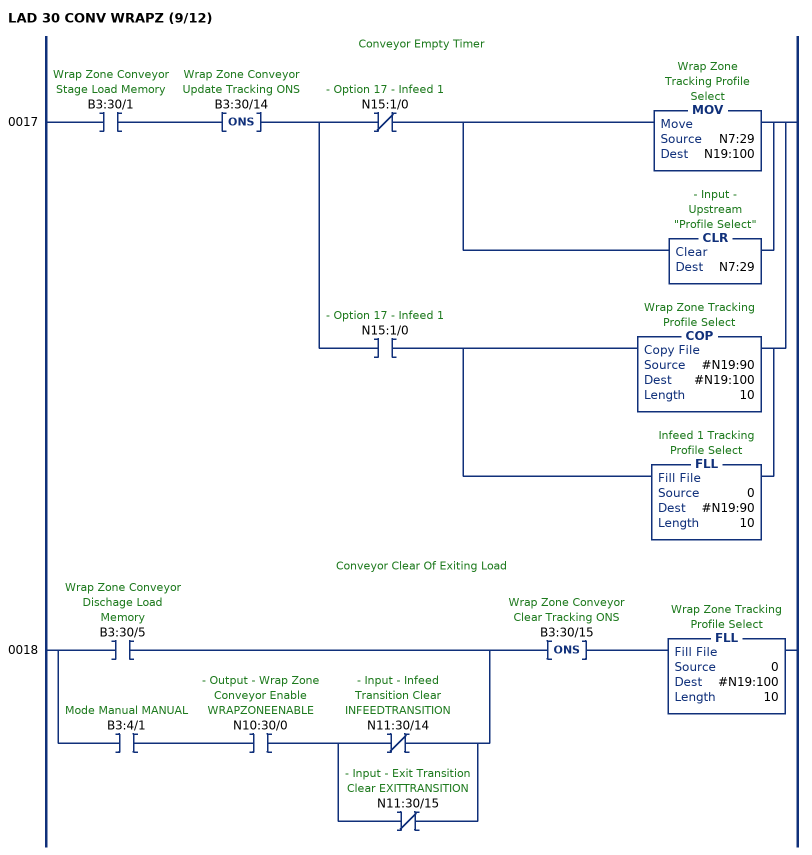
% Rung: 17 %
% Conveyor Empty Timer %
SOR XIC B3:30/1 ONS B3:30/14 BST XIO N15:1/0 BST MOV N7:29 N19:100 NXB CLR N7:29 BND NXB XIC N15:1/0 BST COP #N19:90 #N19:100 10 NXB FLL 0 #N19:90 10 BND BND EOR
%   B3:30/1  "Wrap Zone Conveyor Stage Load Memory" %
%   B3:30/14  "Wrap Zone Conveyor Update Tracking ONS" %
%   N15:1/0  "- Option 17 - Infeed 1" %
%   N7:29  "- Input - Upstream "Profile Select"" %
%   N19:100  "Wrap Zone Tracking Profile Select" %
%   N19:90  "Infeed 1 Tracking Profile Select" %
% Rung: 18 %
% Conveyor Clear Of Exiting Load %
SOR BST XIC B3:30/5 NXB XIC B3:4/1 XIC N10:30/0 BST XIO N11:30/14 NXB XIO N11:30/15 BND BND ONS B3:30/15 FLL 0 #N19:100 10 EOR
%   B3:30/5  "Wrap Zone Conveyor Dischage Load Memory" %
%   B3:4/1  MANUAL  "Mode Manual" %
%   N10:30/0  WRAPZONEENABLE  "- Output - Wrap Zone Conveyor Enable" %
%   N11:30/14  INFEEDTRANSITION  "- Input - Infeed Transition Clear" %
%   N11:30/15  EXITTRANSITION  "- Input - Exit Transition Clear" %
%   B3:30/15  "Wrap Zone Conveyor Clear Tracking ONS" %
%   N19:100  "Wrap Zone Tracking Profile Select" %

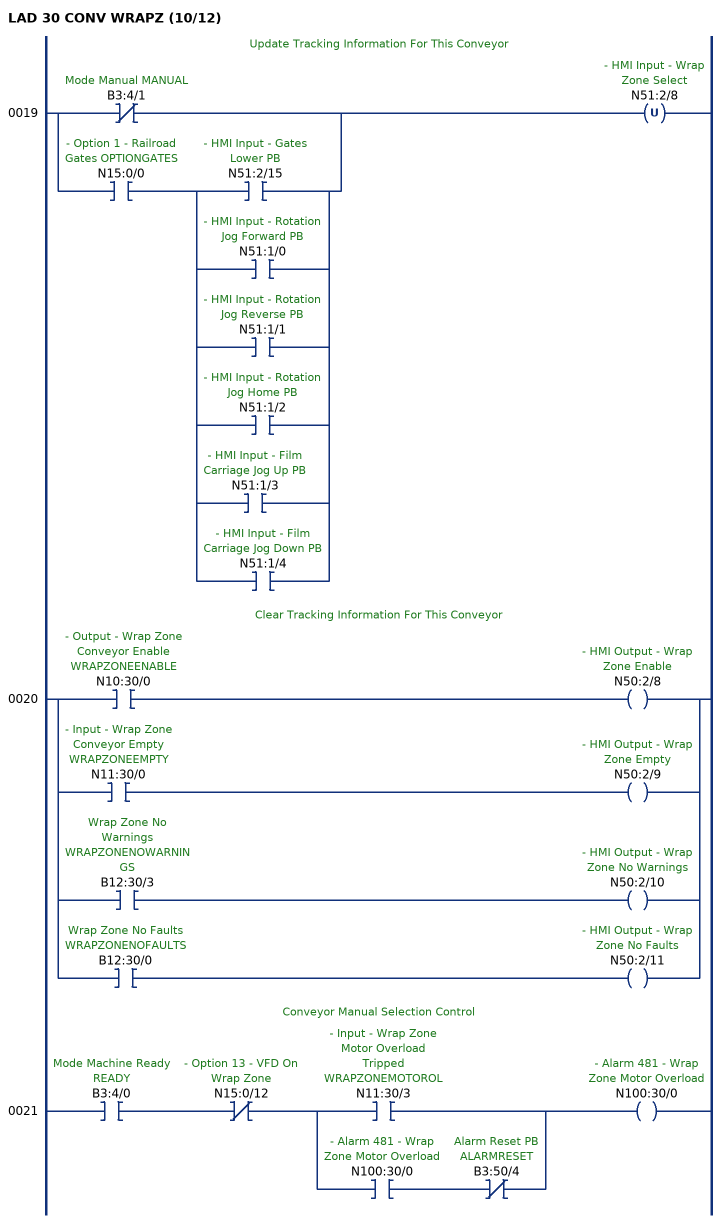
% Rung: 19 %
% Update Tracking Information For This Conveyor %
SOR BST XIO B3:4/1 NXB XIC N15:0/0 BST XIC N51:2/15 NXB XIC N51:1/0 NXB XIC N51:1/1 NXB XIC N51:1/2 NXB XIC N51:1/3 NXB XIC N51:1/4 BND BND OTU N51:2/8 EOR
%   B3:4/1  MANUAL  "Mode Manual" %
%   N15:0/0  OPTIONGATES  "- Option 1 - Railroad Gates" %
%   N51:2/15  "- HMI Input - Gates Lower PB" %
%   N51:1/0  "- HMI Input - Rotation Jog Forward PB" %
%   N51:1/1  "- HMI Input - Rotation Jog Reverse PB" %
%   N51:1/2  "- HMI Input - Rotation Jog Home PB" %
%   N51:1/3  "- HMI Input - Film Carriage Jog Up PB" %
%   N51:1/4  "- HMI Input - Film Carriage Jog Down PB" %
%   N51:2/8  "- HMI Input - Wrap Zone Select" %
% Rung: 20 %
% Clear Tracking Information For This Conveyor %
SOR BST XIC N10:30/0 OTE N50:2/8 NXB XIC N11:30/0 OTE N50:2/9 NXB XIC B12:30/3 OTE N50:2/10 NXB XIC B12:30/0 OTE N50:2/11 BND EOR
%   N10:30/0  WRAPZONEENABLE  "- Output - Wrap Zone Conveyor Enable" %
%   N50:2/8  "- HMI Output - Wrap Zone Enable" %
%   N11:30/0  WRAPZONEEMPTY  "- Input - Wrap Zone Conveyor Empty" %
%   N50:2/9  "- HMI Output - Wrap Zone Empty" %
%   B12:30/3  WRAPZONENOWARNINGS  "Wrap Zone No Warnings" %
%   N50:2/10  "- HMI Output - Wrap Zone No Warnings" %
%   B12:30/0  WRAPZONENOFAULTS  "Wrap Zone No Faults" %
%   N50:2/11  "- HMI Output - Wrap Zone No Faults" %
% Rung: 21 %
% Conveyor Manual Selection Control %
SOR XIC B3:4/0 XIO N15:0/12 BST XIC N11:30/3 NXB XIC N100:30/0 XIO B3:50/4 BND OTE N100:30/0 EOR
%   B3:4/0  READY  "Mode Machine Ready" %
%   N15:0/12  "- Option 13 - VFD On Wrap Zone" %
%   N11:30/3  WRAPZONEMOTOROL  "- Input - Wrap Zone Motor Overload Tripped" %
%   N100:30/0  "- Alarm 481 - Wrap Zone Motor Overload" %
%   B3:50/4  ALARMRESET  "Alarm Reset PB" %

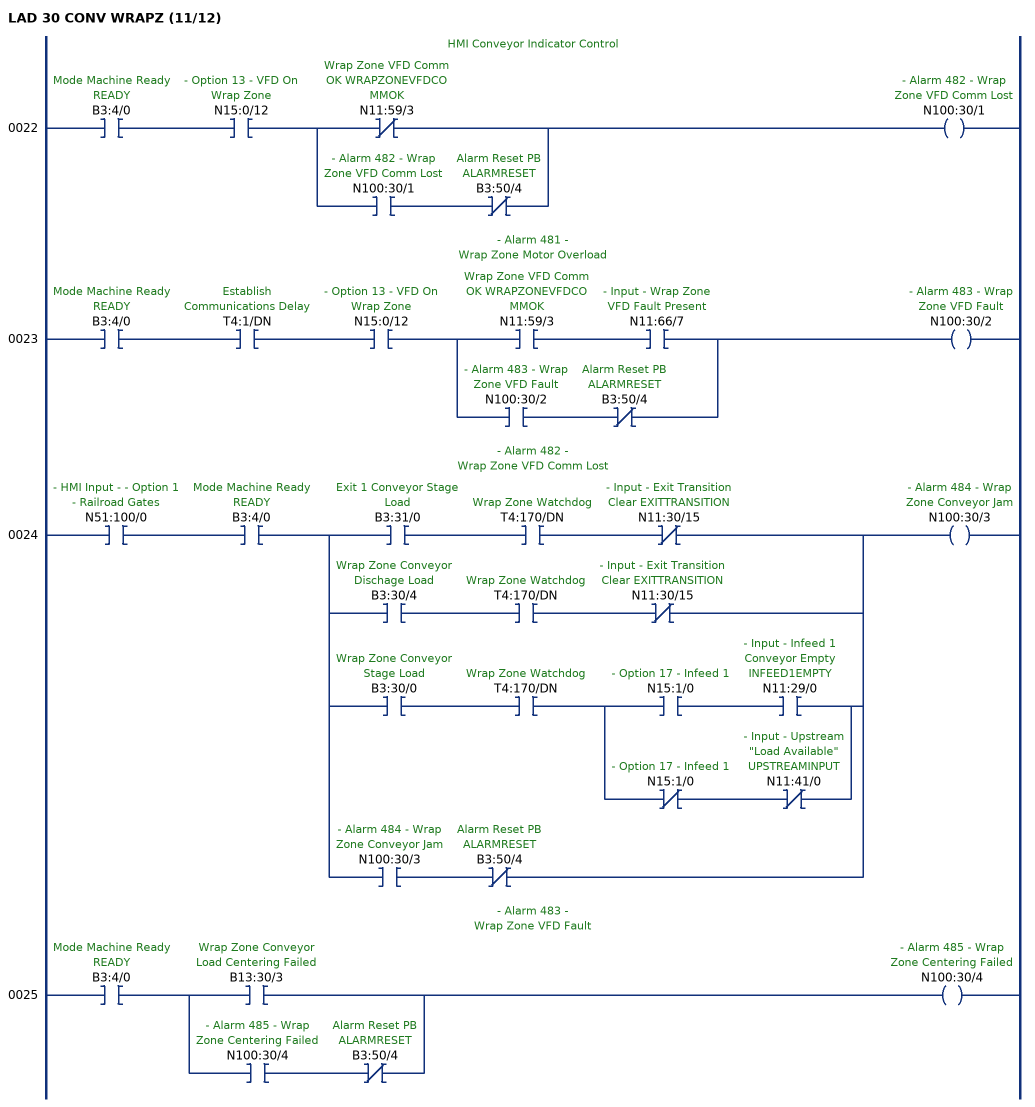
% Rung: 22 %
% HMI Conveyor Indicator Control %
SOR XIC B3:4/0 XIC N15:0/12 BST XIO N11:59/3 NXB XIC N100:30/1 XIO B3:50/4 BND OTE N100:30/1 EOR
%   B3:4/0  READY  "Mode Machine Ready" %
%   N15:0/12  "- Option 13 - VFD On Wrap Zone" %
%   N11:59/3  WRAPZONEVFDCOMMOK  "Wrap Zone VFD Comm OK" %
%   N100:30/1  "- Alarm 482 - Wrap Zone VFD Comm Lost" %
%   B3:50/4  ALARMRESET  "Alarm Reset PB" %
% Rung: 23 %
% - Alarm 481 -
% 
% Wrap Zone Motor Overload %
SOR XIC B3:4/0 XIC T4:1/DN XIC N15:0/12 BST XIC N11:59/3 XIC N11:66/7 NXB XIC N100:30/2 XIO B3:50/4 BND OTE N100:30/2 EOR
%   B3:4/0  READY  "Mode Machine Ready" %
%   T4:1  "Establish Communications Delay" %
%   N15:0/12  "- Option 13 - VFD On Wrap Zone" %
%   N11:59/3  WRAPZONEVFDCOMMOK  "Wrap Zone VFD Comm OK" %
%   N11:66/7  "- Input - Wrap Zone VFD Fault Present" %
%   N100:30/2  "- Alarm 483 - Wrap Zone VFD Fault" %
%   B3:50/4  ALARMRESET  "Alarm Reset PB" %
% Rung: 24 %
% - Alarm 482 -
% 
% Wrap Zone VFD Comm Lost %
SOR XIC N51:100/0 XIC B3:4/0 BST XIC B3:31/0 XIC T4:170/DN XIO N11:30/15 NXB XIC B3:30/4 XIC T4:170/DN XIO N11:30/15 NXB XIC B3:30/0 XIC T4:170/DN BST XIC N15:1/0 XIC N11:29/0 NXB XIO N15:1/0 XIO N11:41/0 BND NXB XIC N100:30/3 XIO B3:50/4 BND OTE N100:30/3 EOR
%   N51:100/0  "- HMI Input - - Option 1 - Railroad Gates" %
%   B3:4/0  READY  "Mode Machine Ready" %
%   B3:31/0  "Exit 1 Conveyor Stage Load" %
%   T4:170  "Wrap Zone Watchdog" %
%   N11:30/15  EXITTRANSITION  "- Input - Exit Transition Clear" %
%   B3:30/4  "Wrap Zone Conveyor Dischage Load" %
%   B3:30/0  "Wrap Zone Conveyor Stage Load" %
%   N15:1/0  "- Option 17 - Infeed 1" %
%   N11:29/0  INFEED1EMPTY  "- Input - Infeed 1 Conveyor Empty" %
%   N11:41/0  UPSTREAMINPUT  "- Input - Upstream "Load Available"" %
%   N100:30/3  "- Alarm 484 - Wrap Zone Conveyor Jam" %
%   B3:50/4  ALARMRESET  "Alarm Reset PB" %
% Rung: 25 %
% - Alarm 483 -
% 
% Wrap Zone VFD Fault %
SOR XIC B3:4/0 BST XIC B13:30/3 NXB XIC N100:30/4 XIO B3:50/4 BND OTE N100:30/4 EOR
%   B3:4/0  READY  "Mode Machine Ready" %
%   B13:30/3  "Wrap Zone Conveyor Load Centering Failed" %
%   N100:30/4  "- Alarm 485 - Wrap Zone Centering Failed" %
%   B3:50/4  ALARMRESET  "Alarm Reset PB" %

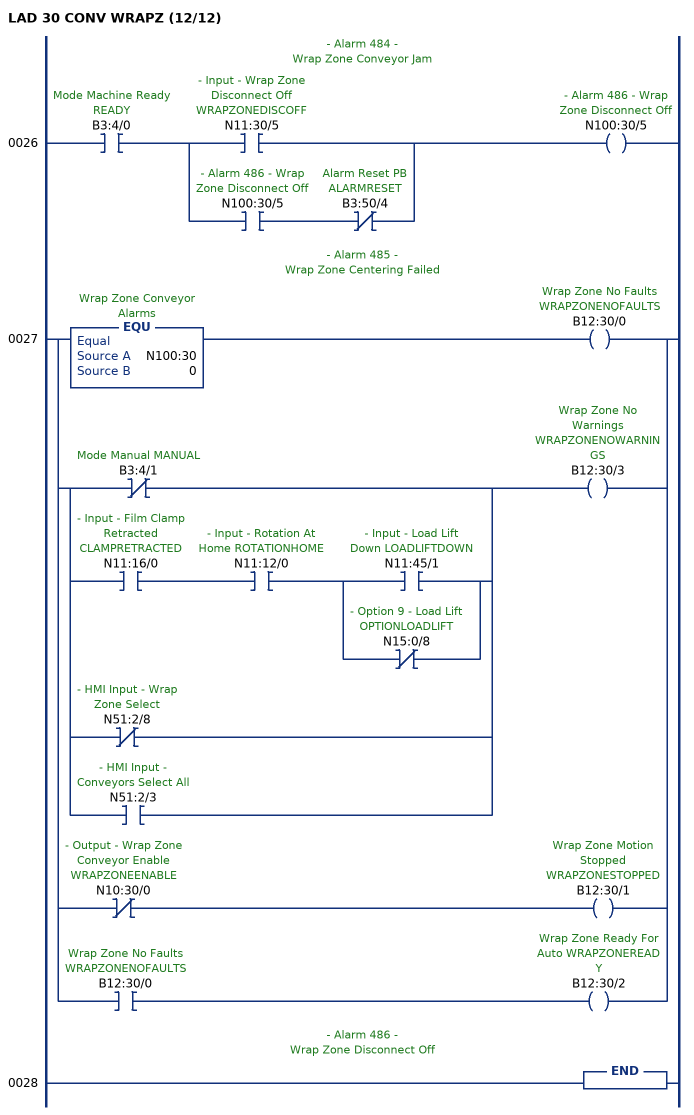
% Rung: 26 %
% - Alarm 484 -
% 
% Wrap Zone Conveyor Jam %
SOR XIC B3:4/0 BST XIC N11:30/5 NXB XIC N100:30/5 XIO B3:50/4 BND OTE N100:30/5 EOR
%   B3:4/0  READY  "Mode Machine Ready" %
%   N11:30/5  WRAPZONEDISCOFF  "- Input - Wrap Zone Disconnect Off" %
%   N100:30/5  "- Alarm 486 - Wrap Zone Disconnect Off" %
%   B3:50/4  ALARMRESET  "Alarm Reset PB" %
% Rung: 27 %
% - Alarm 485 -
% 
% Wrap Zone Centering Failed %
SOR BST EQU N100:30 0 OTE B12:30/0 NXB BST XIO B3:4/1 NXB XIC N11:16/0 XIC N11:12/0 BST XIC N11:45/1 NXB XIO N15:0/8 BND NXB XIO N51:2/8 NXB XIC N51:2/3 BND OTE B12:30/3 NXB XIO N10:30/0 OTE B12:30/1 NXB XIC B12:30/0 OTE B12:30/2 BND EOR
%   N100:30  "Wrap Zone Conveyor Alarms" %
%   B12:30/0  WRAPZONENOFAULTS  "Wrap Zone No Faults" %
%   B3:4/1  MANUAL  "Mode Manual" %
%   N11:16/0  CLAMPRETRACTED  "- Input - Film Clamp Retracted" %
%   N11:12/0  ROTATIONHOME  "- Input - Rotation At Home" %
%   N11:45/1  LOADLIFTDOWN  "- Input - Load Lift Down" %
%   N15:0/8  OPTIONLOADLIFT  "- Option 9 - Load Lift" %
%   N51:2/8  "- HMI Input - Wrap Zone Select" %
%   N51:2/3  "- HMI Input - Conveyors Select All" %
%   B12:30/3  WRAPZONENOWARNINGS  "Wrap Zone No Warnings" %
%   N10:30/0  WRAPZONEENABLE  "- Output - Wrap Zone Conveyor Enable" %
%   B12:30/1  WRAPZONESTOPPED  "Wrap Zone Motion Stopped" %
%   B12:30/2  WRAPZONEREADY  "Wrap Zone Ready For Auto" %
% Rung: 28 %
% - Alarm 486 -
% 
% Wrap Zone Disconnect Off %
SOR END EOR

LADDER 31 "CONV EX 1"
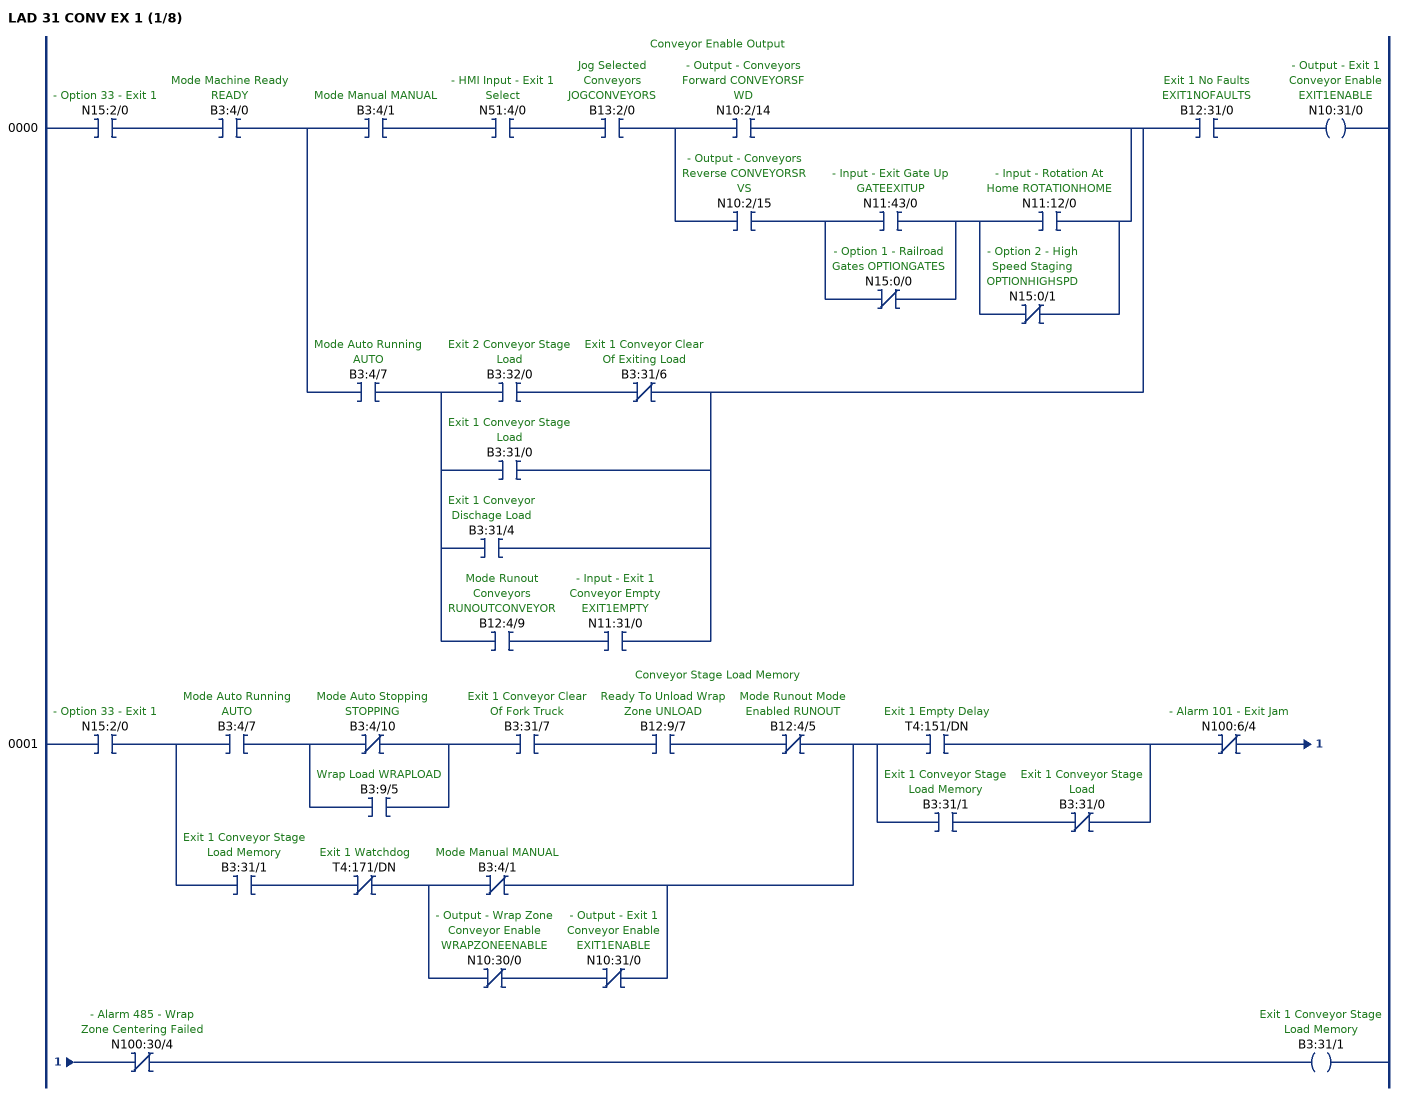
% Rung: 0 %
% Conveyor Enable Output %
SOR XIC N15:2/0 XIC B3:4/0 BST XIC B3:4/1 XIC N51:4/0 XIC B13:2/0 BST XIC N10:2/14 NXB XIC N10:2/15 BST XIC N11:43/0 NXB XIO N15:0/0 BND BST XIC N11:12/0 NXB XIO N15:0/1 BND BND NXB XIC B3:4/7 BST XIC B3:32/0 XIO B3:31/6 NXB XIC B3:31/0 NXB XIC B3:31/4 NXB XIC B12:4/9 XIC N11:31/0 BND BND XIC B12:31/0 OTE N10:31/0 EOR
%   N15:2/0  "- Option 33 - Exit 1" %
%   B3:4/0  READY  "Mode Machine Ready" %
%   B3:4/1  MANUAL  "Mode Manual" %
%   N51:4/0  "- HMI Input - Exit 1 Select" %
%   B13:2/0  JOGCONVEYORS  "Jog Selected Conveyors" %
%   N10:2/14  CONVEYORSFWD  "- Output - Conveyors Forward" %
%   N10:2/15  CONVEYORSRVS  "- Output - Conveyors Reverse" %
%   N11:43/0  GATEEXITUP  "- Input - Exit Gate Up" %
%   N15:0/0  OPTIONGATES  "- Option 1 - Railroad Gates" %
%   N11:12/0  ROTATIONHOME  "- Input - Rotation At Home" %
%   N15:0/1  OPTIONHIGHSPD  "- Option 2 - High Speed Staging" %
%   B3:4/7  AUTO  "Mode Auto Running" %
%   B3:32/0  "Exit 2 Conveyor Stage Load" %
%   B3:31/6  "Exit 1 Conveyor Clear Of Exiting Load" %
%   B3:31/0  "Exit 1 Conveyor Stage Load" %
%   B3:31/4  "Exit 1 Conveyor Dischage Load" %
%   B12:4/9  RUNOUTCONVEYOR  "Mode Runout Conveyors" %
%   N11:31/0  EXIT1EMPTY  "- Input - Exit 1 Conveyor Empty" %
%   B12:31/0  EXIT1NOFAULTS  "Exit 1 No Faults" %
%   N10:31/0  EXIT1ENABLE  "- Output - Exit 1 Conveyor Enable" %
% Rung: 1 %
% Conveyor Stage Load Memory %
SOR XIC N15:2/0 BST XIC B3:4/7 BST XIO B3:4/10 NXB XIC B3:9/5 BND XIC B3:31/7 XIC B12:9/7 XIO B12:4/5 NXB XIC B3:31/1 XIO T4:171/DN BST XIO B3:4/1 NXB XIO N10:30/0 XIO N10:31/0 BND BND BST XIC T4:151/DN NXB XIC B3:31/1 XIO B3:31/0 BND XIO N100:6/4 XIO N100:30/4 OTE B3:31/1 EOR
%   N15:2/0  "- Option 33 - Exit 1" %
%   B3:4/7  AUTO  "Mode Auto Running" %
%   B3:4/10  STOPPING  "Mode Auto Stopping" %
%   B3:9/5  WRAPLOAD  "Wrap Load" %
%   B3:31/7  "Exit 1 Conveyor Clear Of Fork Truck" %
%   B12:9/7  UNLOAD  "Ready To Unload Wrap Zone" %
%   B12:4/5  RUNOUT  "Mode Runout Mode Enabled" %
%   B3:31/1  "Exit 1 Conveyor Stage Load Memory" %
%   T4:171  "Exit 1 Watchdog" %
%   B3:4/1  MANUAL  "Mode Manual" %
%   N10:30/0  WRAPZONEENABLE  "- Output - Wrap Zone Conveyor Enable" %
%   N10:31/0  EXIT1ENABLE  "- Output - Exit 1 Conveyor Enable" %
%   T4:151  "Exit 1 Empty Delay" %
%   B3:31/0  "Exit 1 Conveyor Stage Load" %
%   N100:6/4  "- Alarm 101 - Exit Jam" %
%   N100:30/4  "- Alarm 485 - Wrap Zone Centering Failed" %

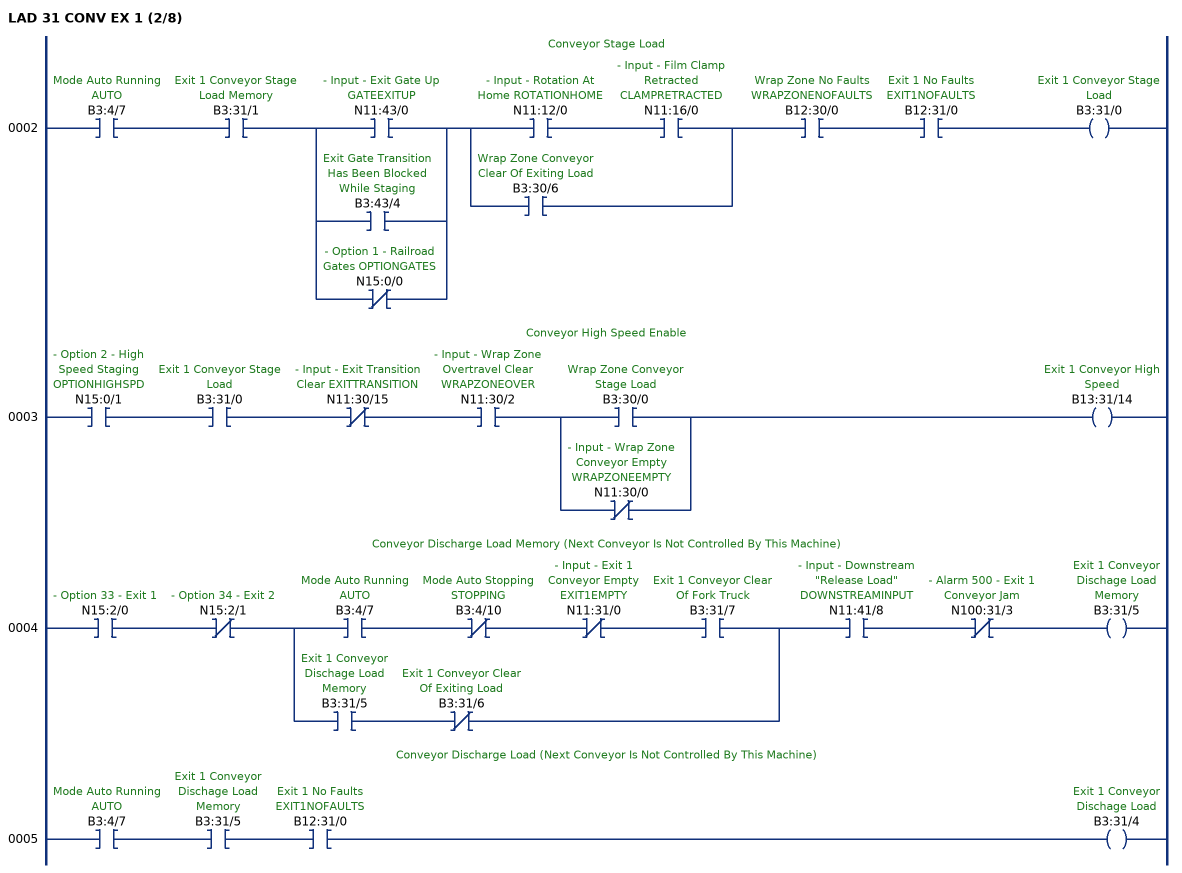
% Rung: 2 %
% Conveyor Stage Load %
SOR XIC B3:4/7 XIC B3:31/1 BST XIC N11:43/0 NXB XIC B3:43/4 NXB XIO N15:0/0 BND BST XIC N11:12/0 XIC N11:16/0 NXB XIC B3:30/6 BND XIC B12:30/0 XIC B12:31/0 OTE B3:31/0 EOR
%   B3:4/7  AUTO  "Mode Auto Running" %
%   B3:31/1  "Exit 1 Conveyor Stage Load Memory" %
%   N11:43/0  GATEEXITUP  "- Input - Exit Gate Up" %
%   B3:43/4  "Exit Gate Transition Has Been Blocked While Staging" %
%   N15:0/0  OPTIONGATES  "- Option 1 - Railroad Gates" %
%   N11:12/0  ROTATIONHOME  "- Input - Rotation At Home" %
%   N11:16/0  CLAMPRETRACTED  "- Input - Film Clamp Retracted" %
%   B3:30/6  "Wrap Zone Conveyor Clear Of Exiting Load" %
%   B12:30/0  WRAPZONENOFAULTS  "Wrap Zone No Faults" %
%   B12:31/0  EXIT1NOFAULTS  "Exit 1 No Faults" %
%   B3:31/0  "Exit 1 Conveyor Stage Load" %
% Rung: 3 %
% Conveyor High Speed Enable %
SOR XIC N15:0/1 XIC B3:31/0 XIO N11:30/15 XIC N11:30/2 BST XIC B3:30/0 NXB XIO N11:30/0 BND OTE B13:31/14 EOR
%   N15:0/1  OPTIONHIGHSPD  "- Option 2 - High Speed Staging" %
%   B3:31/0  "Exit 1 Conveyor Stage Load" %
%   N11:30/15  EXITTRANSITION  "- Input - Exit Transition Clear" %
%   N11:30/2  WRAPZONEOVER  "- Input - Wrap Zone Overtravel Clear" %
%   B3:30/0  "Wrap Zone Conveyor Stage Load" %
%   N11:30/0  WRAPZONEEMPTY  "- Input - Wrap Zone Conveyor Empty" %
%   B13:31/14  "Exit 1 Conveyor High Speed" %
% Rung: 4 %
% Conveyor Discharge Load Memory (Next Conveyor Is Not Controlled By This Machine) %
SOR XIC N15:2/0 XIO N15:2/1 BST XIC B3:4/7 XIO B3:4/10 XIO N11:31/0 XIC B3:31/7 NXB XIC B3:31/5 XIO B3:31/6 BND XIC N11:41/8 XIO N100:31/3 OTE B3:31/5 EOR
%   N15:2/0  "- Option 33 - Exit 1" %
%   N15:2/1  "- Option 34 - Exit 2" %
%   B3:4/7  AUTO  "Mode Auto Running" %
%   B3:4/10  STOPPING  "Mode Auto Stopping" %
%   N11:31/0  EXIT1EMPTY  "- Input - Exit 1 Conveyor Empty" %
%   B3:31/7  "Exit 1 Conveyor Clear Of Fork Truck" %
%   B3:31/5  "Exit 1 Conveyor Dischage Load Memory" %
%   B3:31/6  "Exit 1 Conveyor Clear Of Exiting Load" %
%   N11:41/8  DOWNSTREAMINPUT  "- Input - Downstream "Release Load"" %
%   N100:31/3  "- Alarm 500 - Exit 1 Conveyor Jam" %
% Rung: 5 %
% Conveyor Discharge Load (Next Conveyor Is Not Controlled By This Machine) %
SOR XIC B3:4/7 XIC B3:31/5 XIC B12:31/0 OTE B3:31/4 EOR
%   B3:4/7  AUTO  "Mode Auto Running" %
%   B3:31/5  "Exit 1 Conveyor Dischage Load Memory" %
%   B12:31/0  EXIT1NOFAULTS  "Exit 1 No Faults" %
%   B3:31/4  "Exit 1 Conveyor Dischage Load" %

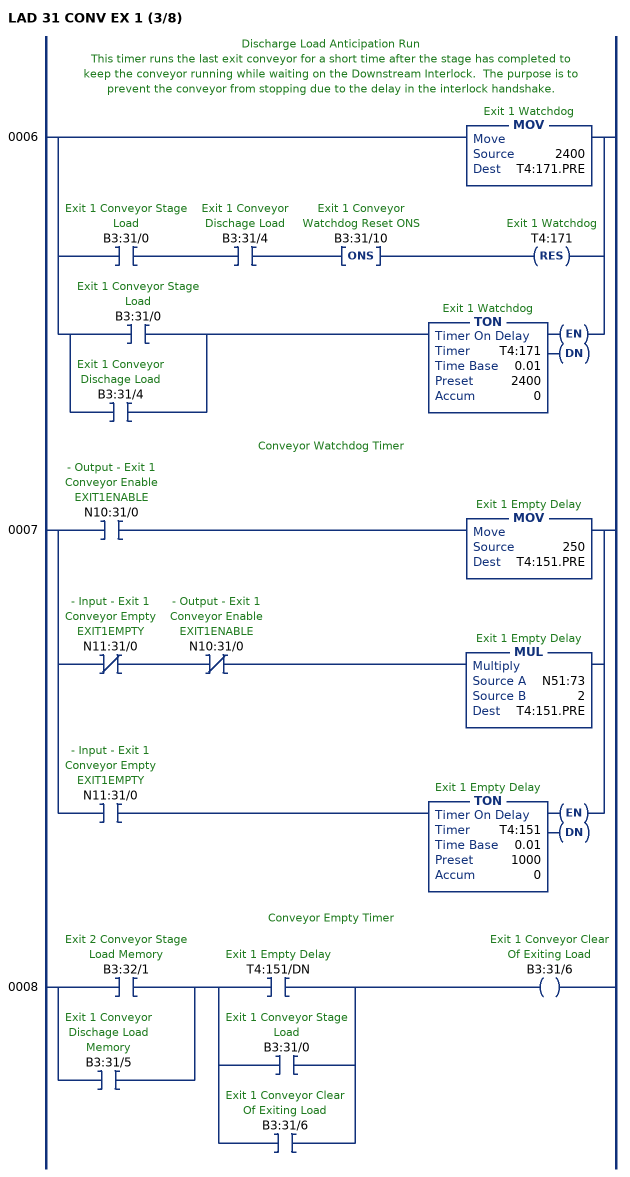
% Rung: 6 %
% Discharge Load Anticipation Run
% 
% This timer runs the last exit conveyor for a short time after the stage has completed to keep the conveyor running while waiting on the Downstream Interlock.  The purpose is to prevent the conveyor from stopping due to the delay in the interlock handshake. %
SOR BST MOV 2400 T4:171.PRE NXB XIC B3:31/0 XIC B3:31/4 ONS B3:31/10 RES T4:171 NXB BST XIC B3:31/0 NXB XIC B3:31/4 BND TON T4:171 0.01 2400 0 BND EOR
%   T4:171  "Exit 1 Watchdog" %
%   B3:31/0  "Exit 1 Conveyor Stage Load" %
%   B3:31/4  "Exit 1 Conveyor Dischage Load" %
%   B3:31/10  "Exit 1 Conveyor Watchdog Reset ONS" %
% Rung: 7 %
% Conveyor Watchdog Timer %
SOR BST XIC N10:31/0 MOV 250 T4:151.PRE NXB XIO N11:31/0 XIO N10:31/0 MUL N51:73 2 T4:151.PRE NXB XIC N11:31/0 TON T4:151 0.01 1000 0 BND EOR
%   N10:31/0  EXIT1ENABLE  "- Output - Exit 1 Conveyor Enable" %
%   T4:151  "Exit 1 Empty Delay" %
%   N11:31/0  EXIT1EMPTY  "- Input - Exit 1 Conveyor Empty" %
%   N51:73  "- HMI Input - Preset Truck Clear" %
% Rung: 8 %
% Conveyor Empty Timer %
SOR BST XIC B3:32/1 NXB XIC B3:31/5 BND BST XIC T4:151/DN NXB XIC B3:31/0 NXB XIC B3:31/6 BND OTE B3:31/6 EOR
%   B3:32/1  "Exit 2 Conveyor Stage Load Memory" %
%   B3:31/5  "Exit 1 Conveyor Dischage Load Memory" %
%   T4:151  "Exit 1 Empty Delay" %
%   B3:31/0  "Exit 1 Conveyor Stage Load" %
%   B3:31/6  "Exit 1 Conveyor Clear Of Exiting Load" %

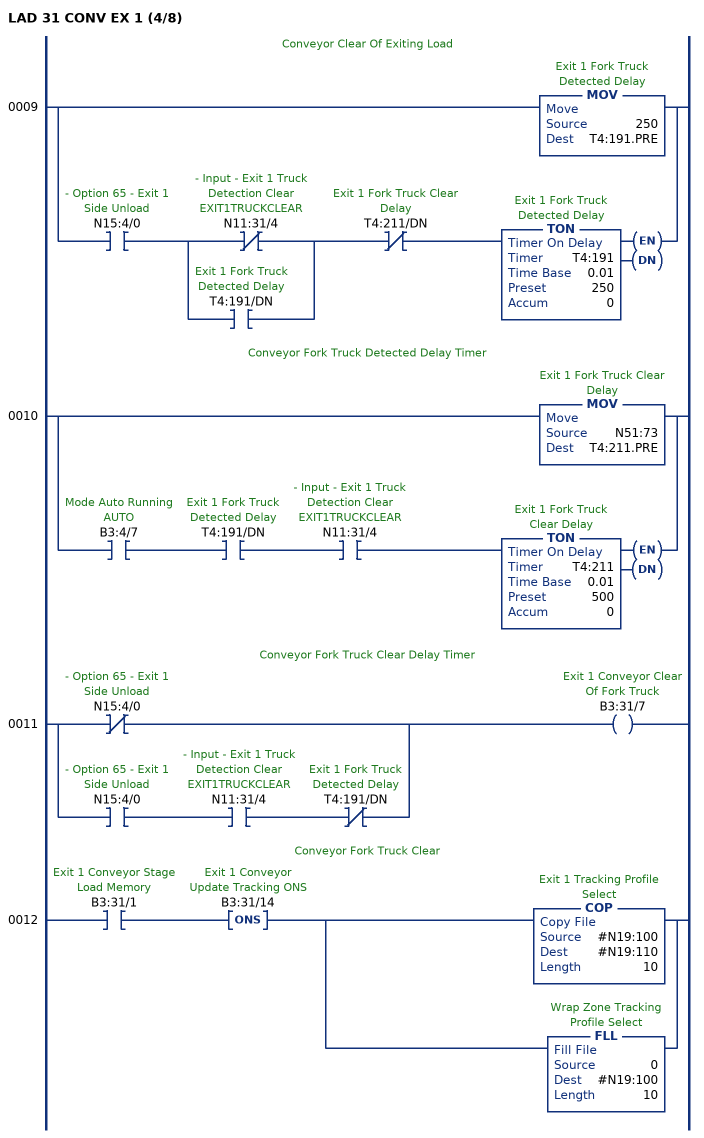
% Rung: 9 %
% Conveyor Clear Of Exiting Load %
SOR BST MOV 250 T4:191.PRE NXB XIC N15:4/0 BST XIO N11:31/4 NXB XIC T4:191/DN BND XIO T4:211/DN TON T4:191 0.01 250 0 BND EOR
%   T4:191  "Exit 1 Fork Truck Detected Delay" %
%   N15:4/0  "- Option 65 - Exit 1 Side Unload" %
%   N11:31/4  EXIT1TRUCKCLEAR  "- Input - Exit 1 Truck Detection Clear" %
%   T4:211  "Exit 1 Fork Truck Clear Delay" %
% Rung: 10 %
% Conveyor Fork Truck Detected Delay Timer %
SOR BST MOV N51:73 T4:211.PRE NXB XIC B3:4/7 XIC T4:191/DN XIC N11:31/4 TON T4:211 0.01 500 0 BND EOR
%   N51:73  "- HMI Input - Preset Truck Clear" %
%   T4:211  "Exit 1 Fork Truck Clear Delay" %
%   B3:4/7  AUTO  "Mode Auto Running" %
%   T4:191  "Exit 1 Fork Truck Detected Delay" %
%   N11:31/4  EXIT1TRUCKCLEAR  "- Input - Exit 1 Truck Detection Clear" %
% Rung: 11 %
% Conveyor Fork Truck Clear Delay Timer %
SOR BST XIO N15:4/0 NXB XIC N15:4/0 XIC N11:31/4 XIO T4:191/DN BND OTE B3:31/7 EOR
%   N15:4/0  "- Option 65 - Exit 1 Side Unload" %
%   N11:31/4  EXIT1TRUCKCLEAR  "- Input - Exit 1 Truck Detection Clear" %
%   T4:191  "Exit 1 Fork Truck Detected Delay" %
%   B3:31/7  "Exit 1 Conveyor Clear Of Fork Truck" %
% Rung: 12 %
% Conveyor Fork Truck Clear %
SOR XIC B3:31/1 ONS B3:31/14 BST COP #N19:100 #N19:110 10 NXB FLL 0 #N19:100 10 BND EOR
%   B3:31/1  "Exit 1 Conveyor Stage Load Memory" %
%   B3:31/14  "Exit 1 Conveyor Update Tracking ONS" %
%   N19:100  "Wrap Zone Tracking Profile Select" %
%   N19:110  "Exit 1 Tracking Profile Select" %

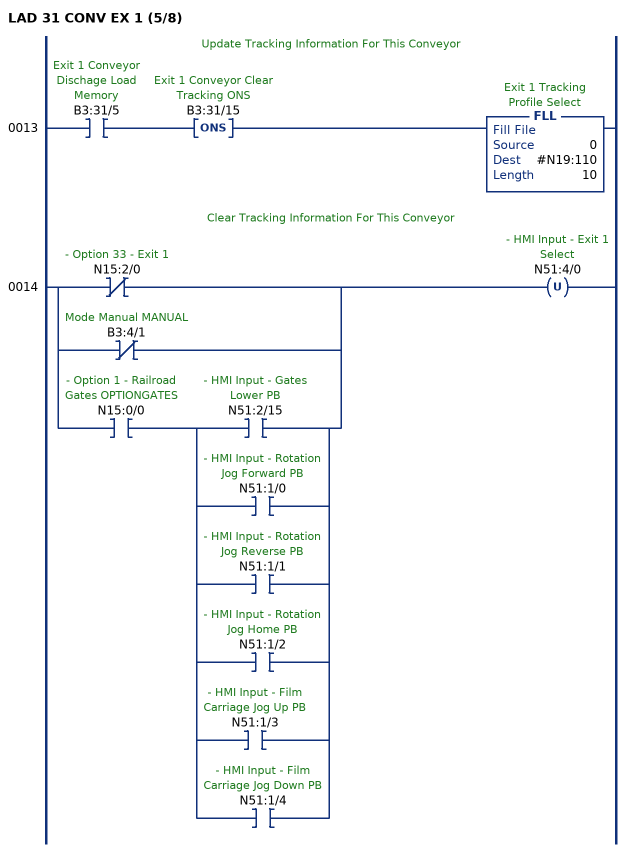
% Rung: 13 %
% Update Tracking Information For This Conveyor %
SOR XIC B3:31/5 ONS B3:31/15 FLL 0 #N19:110 10 EOR
%   B3:31/5  "Exit 1 Conveyor Dischage Load Memory" %
%   B3:31/15  "Exit 1 Conveyor Clear Tracking ONS" %
%   N19:110  "Exit 1 Tracking Profile Select" %
% Rung: 14 %
% Clear Tracking Information For This Conveyor %
SOR BST XIO N15:2/0 NXB XIO B3:4/1 NXB XIC N15:0/0 BST XIC N51:2/15 NXB XIC N51:1/0 NXB XIC N51:1/1 NXB XIC N51:1/2 NXB XIC N51:1/3 NXB XIC N51:1/4 BND BND OTU N51:4/0 EOR
%   N15:2/0  "- Option 33 - Exit 1" %
%   B3:4/1  MANUAL  "Mode Manual" %
%   N15:0/0  OPTIONGATES  "- Option 1 - Railroad Gates" %
%   N51:2/15  "- HMI Input - Gates Lower PB" %
%   N51:1/0  "- HMI Input - Rotation Jog Forward PB" %
%   N51:1/1  "- HMI Input - Rotation Jog Reverse PB" %
%   N51:1/2  "- HMI Input - Rotation Jog Home PB" %
%   N51:1/3  "- HMI Input - Film Carriage Jog Up PB" %
%   N51:1/4  "- HMI Input - Film Carriage Jog Down PB" %
%   N51:4/0  "- HMI Input - Exit 1 Select" %

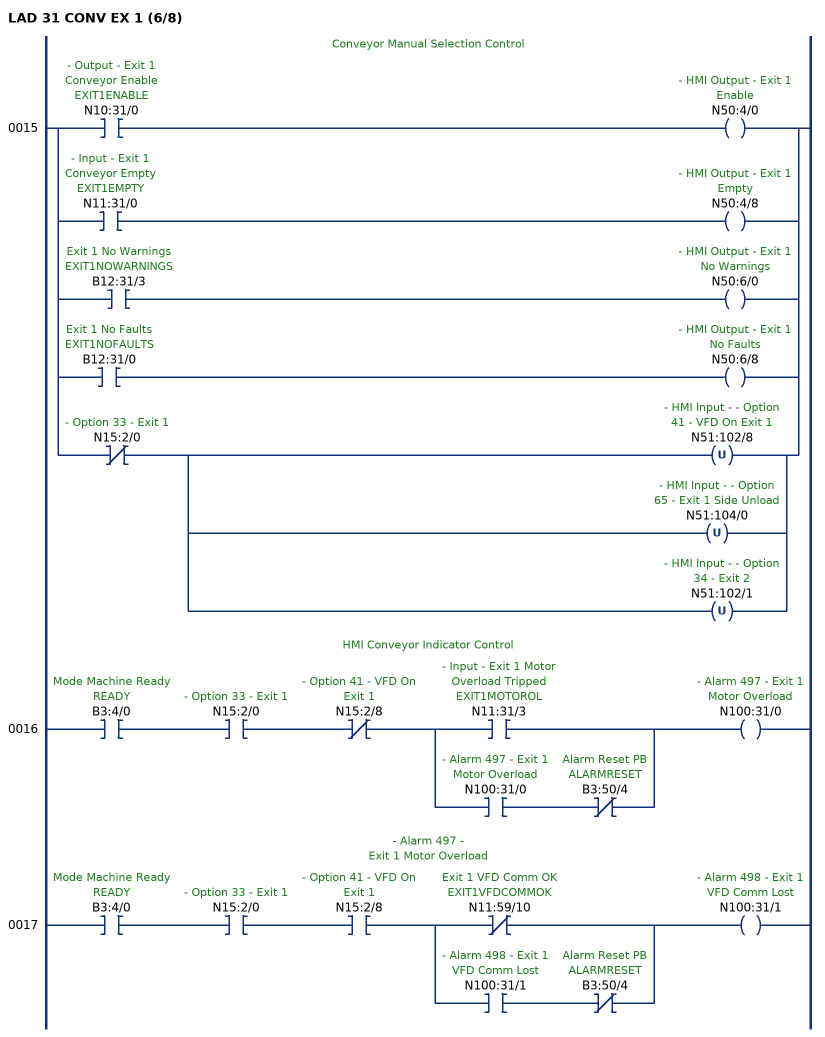
% Rung: 15 %
% Conveyor Manual Selection Control %
SOR BST XIC N10:31/0 OTE N50:4/0 NXB XIC N11:31/0 OTE N50:4/8 NXB XIC B12:31/3 OTE N50:6/0 NXB XIC B12:31/0 OTE N50:6/8 NXB XIO N15:2/0 BST OTU N51:102/8 NXB OTU N51:104/0 NXB OTU N51:102/1 BND BND EOR
%   N10:31/0  EXIT1ENABLE  "- Output - Exit 1 Conveyor Enable" %
%   N50:4/0  "- HMI Output - Exit 1 Enable" %
%   N11:31/0  EXIT1EMPTY  "- Input - Exit 1 Conveyor Empty" %
%   N50:4/8  "- HMI Output - Exit 1 Empty" %
%   B12:31/3  EXIT1NOWARNINGS  "Exit 1 No Warnings" %
%   N50:6/0  "- HMI Output - Exit 1 No Warnings" %
%   B12:31/0  EXIT1NOFAULTS  "Exit 1 No Faults" %
%   N50:6/8  "- HMI Output - Exit 1 No Faults" %
%   N15:2/0  "- Option 33 - Exit 1" %
%   N51:102/8  "- HMI Input - - Option 41 - VFD On Exit 1" %
%   N51:104/0  "- HMI Input - - Option 65 - Exit 1 Side Unload" %
%   N51:102/1  "- HMI Input - - Option 34 - Exit 2" %
% Rung: 16 %
% HMI Conveyor Indicator Control %
SOR XIC B3:4/0 XIC N15:2/0 XIO N15:2/8 BST XIC N11:31/3 NXB XIC N100:31/0 XIO B3:50/4 BND OTE N100:31/0 EOR
%   B3:4/0  READY  "Mode Machine Ready" %
%   N15:2/0  "- Option 33 - Exit 1" %
%   N15:2/8  "- Option 41 - VFD On Exit 1" %
%   N11:31/3  EXIT1MOTOROL  "- Input - Exit 1 Motor Overload Tripped" %
%   N100:31/0  "- Alarm 497 - Exit 1 Motor Overload" %
%   B3:50/4  ALARMRESET  "Alarm Reset PB" %
% Rung: 17 %
% - Alarm 497 -
% 
% Exit 1 Motor Overload %
SOR XIC B3:4/0 XIC N15:2/0 XIC N15:2/8 BST XIO N11:59/10 NXB XIC N100:31/1 XIO B3:50/4 BND OTE N100:31/1 EOR
%   B3:4/0  READY  "Mode Machine Ready" %
%   N15:2/0  "- Option 33 - Exit 1" %
%   N15:2/8  "- Option 41 - VFD On Exit 1" %
%   N11:59/10  EXIT1VFDCOMMOK  "Exit 1 VFD Comm OK" %
%   N100:31/1  "- Alarm 498 - Exit 1 VFD Comm Lost" %
%   B3:50/4  ALARMRESET  "Alarm Reset PB" %

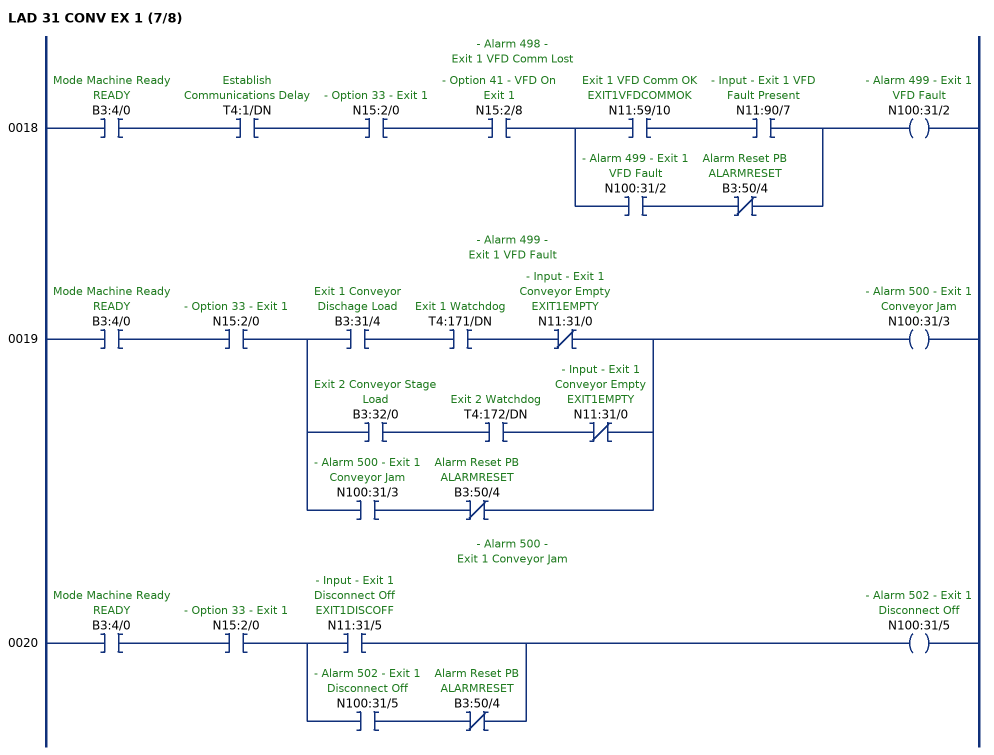
% Rung: 18 %
% - Alarm 498 -
% 
% Exit 1 VFD Comm Lost %
SOR XIC B3:4/0 XIC T4:1/DN XIC N15:2/0 XIC N15:2/8 BST XIC N11:59/10 XIC N11:90/7 NXB XIC N100:31/2 XIO B3:50/4 BND OTE N100:31/2 EOR
%   B3:4/0  READY  "Mode Machine Ready" %
%   T4:1  "Establish Communications Delay" %
%   N15:2/0  "- Option 33 - Exit 1" %
%   N15:2/8  "- Option 41 - VFD On Exit 1" %
%   N11:59/10  EXIT1VFDCOMMOK  "Exit 1 VFD Comm OK" %
%   N11:90/7  "- Input - Exit 1 VFD Fault Present" %
%   N100:31/2  "- Alarm 499 - Exit 1 VFD Fault" %
%   B3:50/4  ALARMRESET  "Alarm Reset PB" %
% Rung: 19 %
% - Alarm 499 -
% 
% Exit 1 VFD Fault %
SOR XIC B3:4/0 XIC N15:2/0 BST XIC B3:31/4 XIC T4:171/DN XIO N11:31/0 NXB XIC B3:32/0 XIC T4:172/DN XIO N11:31/0 NXB XIC N100:31/3 XIO B3:50/4 BND OTE N100:31/3 EOR
%   B3:4/0  READY  "Mode Machine Ready" %
%   N15:2/0  "- Option 33 - Exit 1" %
%   B3:31/4  "Exit 1 Conveyor Dischage Load" %
%   T4:171  "Exit 1 Watchdog" %
%   N11:31/0  EXIT1EMPTY  "- Input - Exit 1 Conveyor Empty" %
%   B3:32/0  "Exit 2 Conveyor Stage Load" %
%   T4:172  "Exit 2 Watchdog" %
%   N100:31/3  "- Alarm 500 - Exit 1 Conveyor Jam" %
%   B3:50/4  ALARMRESET  "Alarm Reset PB" %
% Rung: 20 %
% - Alarm 500 -
% 
% Exit 1 Conveyor Jam %
SOR XIC B3:4/0 XIC N15:2/0 BST XIC N11:31/5 NXB XIC N100:31/5 XIO B3:50/4 BND OTE N100:31/5 EOR
%   B3:4/0  READY  "Mode Machine Ready" %
%   N15:2/0  "- Option 33 - Exit 1" %
%   N11:31/5  EXIT1DISCOFF  "- Input - Exit 1 Disconnect Off" %
%   N100:31/5  "- Alarm 502 - Exit 1 Disconnect Off" %
%   B3:50/4  ALARMRESET  "Alarm Reset PB" %

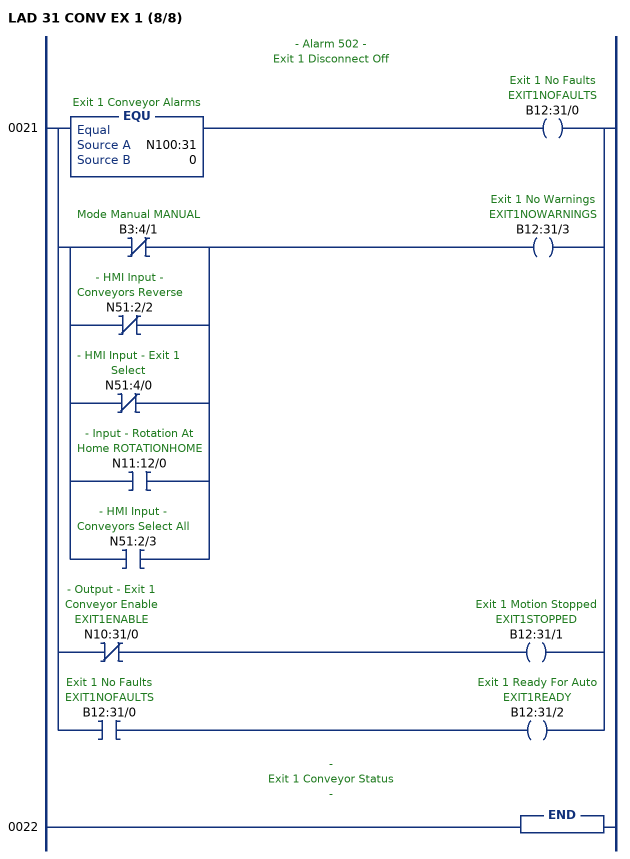
% Rung: 21 %
% - Alarm 502 -
% 
% Exit 1 Disconnect Off %
SOR BST EQU N100:31 0 OTE B12:31/0 NXB BST XIO B3:4/1 NXB XIO N51:2/2 NXB XIO N51:4/0 NXB XIC N11:12/0 NXB XIC N51:2/3 BND OTE B12:31/3 NXB XIO N10:31/0 OTE B12:31/1 NXB XIC B12:31/0 OTE B12:31/2 BND EOR
%   N100:31  "Exit 1 Conveyor Alarms" %
%   B12:31/0  EXIT1NOFAULTS  "Exit 1 No Faults" %
%   B3:4/1  MANUAL  "Mode Manual" %
%   N51:2/2  "- HMI Input - Conveyors Reverse" %
%   N51:4/0  "- HMI Input - Exit 1 Select" %
%   N11:12/0  ROTATIONHOME  "- Input - Rotation At Home" %
%   N51:2/3  "- HMI Input - Conveyors Select All" %
%   B12:31/3  EXIT1NOWARNINGS  "Exit 1 No Warnings" %
%   N10:31/0  EXIT1ENABLE  "- Output - Exit 1 Conveyor Enable" %
%   B12:31/1  EXIT1STOPPED  "Exit 1 Motion Stopped" %
%   B12:31/2  EXIT1READY  "Exit 1 Ready For Auto" %
% Rung: 22 %
% -
% 
% Exit 1 Conveyor Status
% 
% - %
SOR END EOR

LADDER 32 "CONV EX 2"
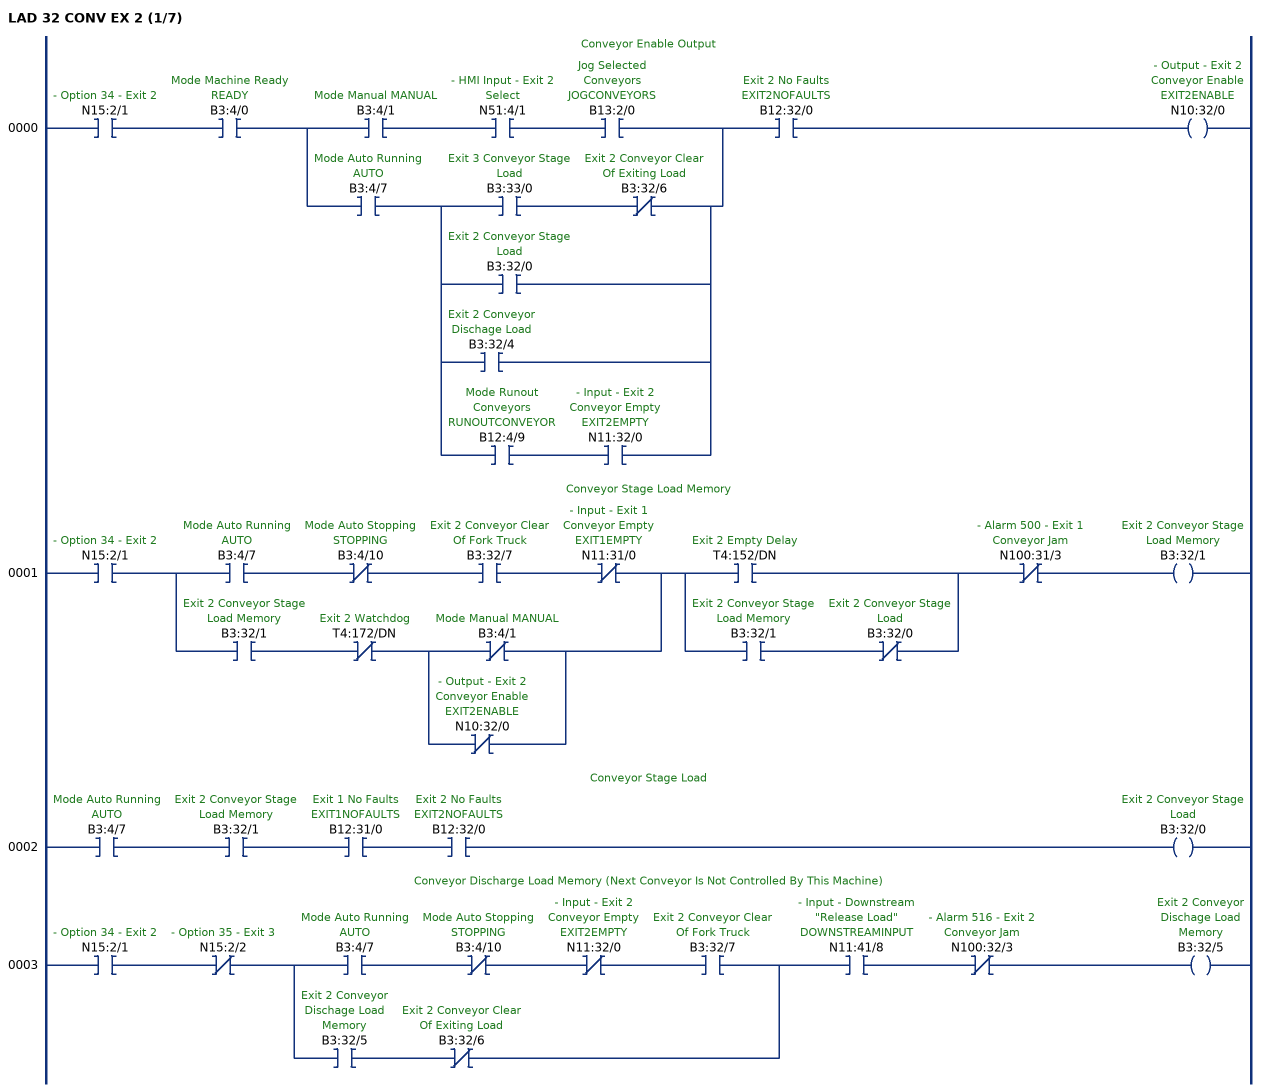
% Rung: 0 %
% Conveyor Enable Output %
SOR XIC N15:2/1 XIC B3:4/0 BST XIC B3:4/1 XIC N51:4/1 XIC B13:2/0 NXB XIC B3:4/7 BST XIC B3:33/0 XIO B3:32/6 NXB XIC B3:32/0 NXB XIC B3:32/4 NXB XIC B12:4/9 XIC N11:32/0 BND BND XIC B12:32/0 OTE N10:32/0 EOR
%   N15:2/1  "- Option 34 - Exit 2" %
%   B3:4/0  READY  "Mode Machine Ready" %
%   B3:4/1  MANUAL  "Mode Manual" %
%   N51:4/1  "- HMI Input - Exit 2 Select" %
%   B13:2/0  JOGCONVEYORS  "Jog Selected Conveyors" %
%   B3:4/7  AUTO  "Mode Auto Running" %
%   B3:33/0  "Exit 3 Conveyor Stage Load" %
%   B3:32/6  "Exit 2 Conveyor Clear Of Exiting Load" %
%   B3:32/0  "Exit 2 Conveyor Stage Load" %
%   B3:32/4  "Exit 2 Conveyor Dischage Load" %
%   B12:4/9  RUNOUTCONVEYOR  "Mode Runout Conveyors" %
%   N11:32/0  EXIT2EMPTY  "- Input - Exit 2 Conveyor Empty" %
%   B12:32/0  EXIT2NOFAULTS  "Exit 2 No Faults" %
%   N10:32/0  EXIT2ENABLE  "- Output - Exit 2 Conveyor Enable" %
% Rung: 1 %
% Conveyor Stage Load Memory %
SOR XIC N15:2/1 BST XIC B3:4/7 XIO B3:4/10 XIC B3:32/7 XIO N11:31/0 NXB XIC B3:32/1 XIO T4:172/DN BST XIO B3:4/1 NXB XIO N10:32/0 BND BND BST XIC T4:152/DN NXB XIC B3:32/1 XIO B3:32/0 BND XIO N100:31/3 OTE B3:32/1 EOR
%   N15:2/1  "- Option 34 - Exit 2" %
%   B3:4/7  AUTO  "Mode Auto Running" %
%   B3:4/10  STOPPING  "Mode Auto Stopping" %
%   B3:32/7  "Exit 2 Conveyor Clear Of Fork Truck" %
%   N11:31/0  EXIT1EMPTY  "- Input - Exit 1 Conveyor Empty" %
%   B3:32/1  "Exit 2 Conveyor Stage Load Memory" %
%   T4:172  "Exit 2 Watchdog" %
%   B3:4/1  MANUAL  "Mode Manual" %
%   N10:32/0  EXIT2ENABLE  "- Output - Exit 2 Conveyor Enable" %
%   T4:152  "Exit 2 Empty Delay" %
%   B3:32/0  "Exit 2 Conveyor Stage Load" %
%   N100:31/3  "- Alarm 500 - Exit 1 Conveyor Jam" %
% Rung: 2 %
% Conveyor Stage Load %
SOR XIC B3:4/7 XIC B3:32/1 XIC B12:31/0 XIC B12:32/0 OTE B3:32/0 EOR
%   B3:4/7  AUTO  "Mode Auto Running" %
%   B3:32/1  "Exit 2 Conveyor Stage Load Memory" %
%   B12:31/0  EXIT1NOFAULTS  "Exit 1 No Faults" %
%   B12:32/0  EXIT2NOFAULTS  "Exit 2 No Faults" %
%   B3:32/0  "Exit 2 Conveyor Stage Load" %
% Rung: 3 %
% Conveyor Discharge Load Memory (Next Conveyor Is Not Controlled By This Machine) %
SOR XIC N15:2/1 XIO N15:2/2 BST XIC B3:4/7 XIO B3:4/10 XIO N11:32/0 XIC B3:32/7 NXB XIC B3:32/5 XIO B3:32/6 BND XIC N11:41/8 XIO N100:32/3 OTE B3:32/5 EOR
%   N15:2/1  "- Option 34 - Exit 2" %
%   N15:2/2  "- Option 35 - Exit 3" %
%   B3:4/7  AUTO  "Mode Auto Running" %
%   B3:4/10  STOPPING  "Mode Auto Stopping" %
%   N11:32/0  EXIT2EMPTY  "- Input - Exit 2 Conveyor Empty" %
%   B3:32/7  "Exit 2 Conveyor Clear Of Fork Truck" %
%   B3:32/5  "Exit 2 Conveyor Dischage Load Memory" %
%   B3:32/6  "Exit 2 Conveyor Clear Of Exiting Load" %
%   N11:41/8  DOWNSTREAMINPUT  "- Input - Downstream "Release Load"" %
%   N100:32/3  "- Alarm 516 - Exit 2 Conveyor Jam" %

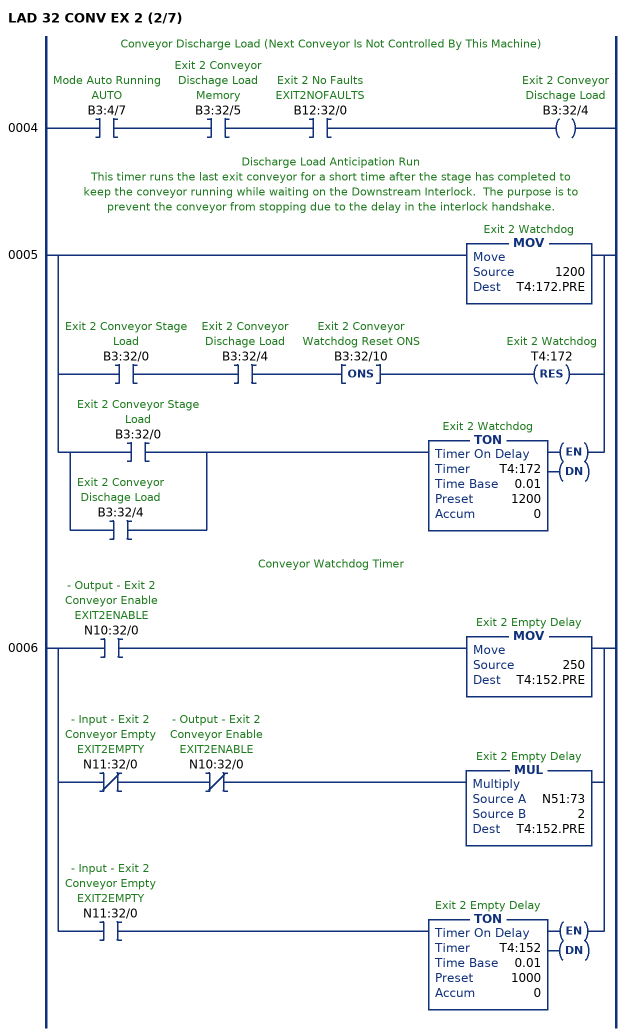
% Rung: 4 %
% Conveyor Discharge Load (Next Conveyor Is Not Controlled By This Machine) %
SOR XIC B3:4/7 XIC B3:32/5 XIC B12:32/0 OTE B3:32/4 EOR
%   B3:4/7  AUTO  "Mode Auto Running" %
%   B3:32/5  "Exit 2 Conveyor Dischage Load Memory" %
%   B12:32/0  EXIT2NOFAULTS  "Exit 2 No Faults" %
%   B3:32/4  "Exit 2 Conveyor Dischage Load" %
% Rung: 5 %
% Discharge Load Anticipation Run
% 
% This timer runs the last exit conveyor for a short time after the stage has completed to keep the conveyor running while waiting on the Downstream Interlock.  The purpose is to prevent the conveyor from stopping due to the delay in the interlock handshake. %
SOR BST MOV 1200 T4:172.PRE NXB XIC B3:32/0 XIC B3:32/4 ONS B3:32/10 RES T4:172 NXB BST XIC B3:32/0 NXB XIC B3:32/4 BND TON T4:172 0.01 1200 0 BND EOR
%   T4:172  "Exit 2 Watchdog" %
%   B3:32/0  "Exit 2 Conveyor Stage Load" %
%   B3:32/4  "Exit 2 Conveyor Dischage Load" %
%   B3:32/10  "Exit 2 Conveyor Watchdog Reset ONS" %
% Rung: 6 %
% Conveyor Watchdog Timer %
SOR BST XIC N10:32/0 MOV 250 T4:152.PRE NXB XIO N11:32/0 XIO N10:32/0 MUL N51:73 2 T4:152.PRE NXB XIC N11:32/0 TON T4:152 0.01 1000 0 BND EOR
%   N10:32/0  EXIT2ENABLE  "- Output - Exit 2 Conveyor Enable" %
%   T4:152  "Exit 2 Empty Delay" %
%   N11:32/0  EXIT2EMPTY  "- Input - Exit 2 Conveyor Empty" %
%   N51:73  "- HMI Input - Preset Truck Clear" %

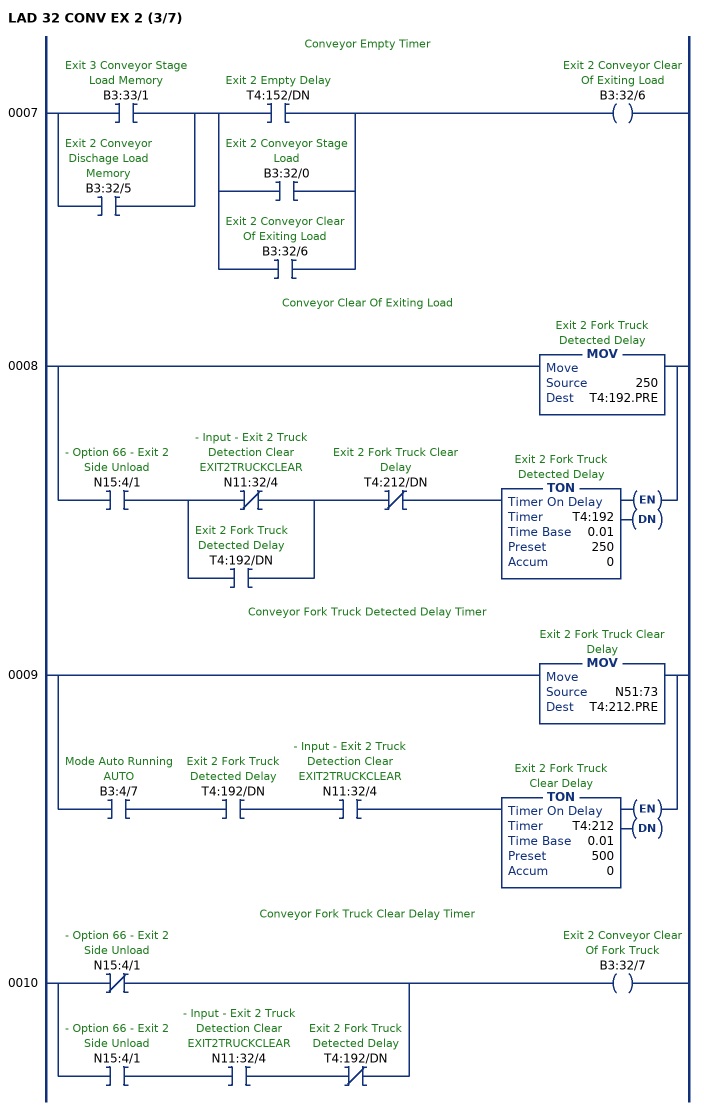
% Rung: 7 %
% Conveyor Empty Timer %
SOR BST XIC B3:33/1 NXB XIC B3:32/5 BND BST XIC T4:152/DN NXB XIC B3:32/0 NXB XIC B3:32/6 BND OTE B3:32/6 EOR
%   B3:33/1  "Exit 3 Conveyor Stage Load Memory" %
%   B3:32/5  "Exit 2 Conveyor Dischage Load Memory" %
%   T4:152  "Exit 2 Empty Delay" %
%   B3:32/0  "Exit 2 Conveyor Stage Load" %
%   B3:32/6  "Exit 2 Conveyor Clear Of Exiting Load" %
% Rung: 8 %
% Conveyor Clear Of Exiting Load %
SOR BST MOV 250 T4:192.PRE NXB XIC N15:4/1 BST XIO N11:32/4 NXB XIC T4:192/DN BND XIO T4:212/DN TON T4:192 0.01 250 0 BND EOR
%   T4:192  "Exit 2 Fork Truck Detected Delay" %
%   N15:4/1  "- Option 66 - Exit 2 Side Unload" %
%   N11:32/4  EXIT2TRUCKCLEAR  "- Input - Exit 2 Truck Detection Clear" %
%   T4:212  "Exit 2 Fork Truck Clear Delay" %
% Rung: 9 %
% Conveyor Fork Truck Detected Delay Timer %
SOR BST MOV N51:73 T4:212.PRE NXB XIC B3:4/7 XIC T4:192/DN XIC N11:32/4 TON T4:212 0.01 500 0 BND EOR
%   N51:73  "- HMI Input - Preset Truck Clear" %
%   T4:212  "Exit 2 Fork Truck Clear Delay" %
%   B3:4/7  AUTO  "Mode Auto Running" %
%   T4:192  "Exit 2 Fork Truck Detected Delay" %
%   N11:32/4  EXIT2TRUCKCLEAR  "- Input - Exit 2 Truck Detection Clear" %
% Rung: 10 %
% Conveyor Fork Truck Clear Delay Timer %
SOR BST XIO N15:4/1 NXB XIC N15:4/1 XIC N11:32/4 XIO T4:192/DN BND OTE B3:32/7 EOR
%   N15:4/1  "- Option 66 - Exit 2 Side Unload" %
%   N11:32/4  EXIT2TRUCKCLEAR  "- Input - Exit 2 Truck Detection Clear" %
%   T4:192  "Exit 2 Fork Truck Detected Delay" %
%   B3:32/7  "Exit 2 Conveyor Clear Of Fork Truck" %

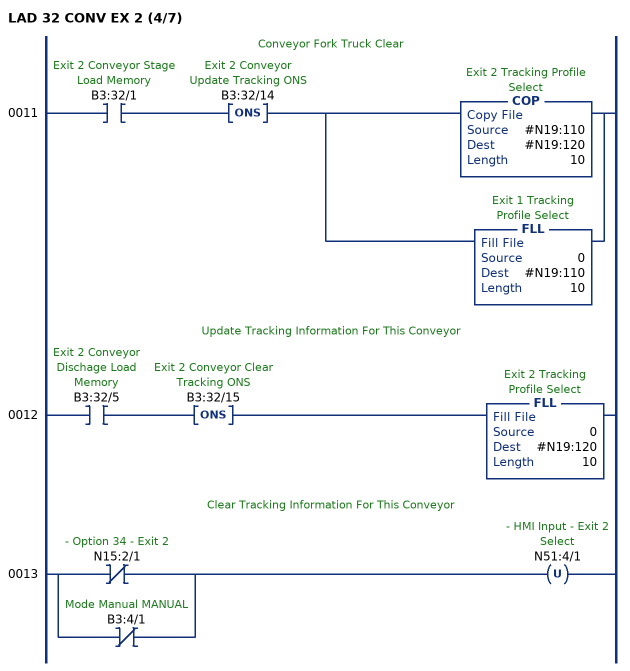
% Rung: 11 %
% Conveyor Fork Truck Clear %
SOR XIC B3:32/1 ONS B3:32/14 BST COP #N19:110 #N19:120 10 NXB FLL 0 #N19:110 10 BND EOR
%   B3:32/1  "Exit 2 Conveyor Stage Load Memory" %
%   B3:32/14  "Exit 2 Conveyor Update Tracking ONS" %
%   N19:110  "Exit 1 Tracking Profile Select" %
%   N19:120  "Exit 2 Tracking Profile Select" %
% Rung: 12 %
% Update Tracking Information For This Conveyor %
SOR XIC B3:32/5 ONS B3:32/15 FLL 0 #N19:120 10 EOR
%   B3:32/5  "Exit 2 Conveyor Dischage Load Memory" %
%   B3:32/15  "Exit 2 Conveyor Clear Tracking ONS" %
%   N19:120  "Exit 2 Tracking Profile Select" %
% Rung: 13 %
% Clear Tracking Information For This Conveyor %
SOR BST XIO N15:2/1 NXB XIO B3:4/1 BND OTU N51:4/1 EOR
%   N15:2/1  "- Option 34 - Exit 2" %
%   B3:4/1  MANUAL  "Mode Manual" %
%   N51:4/1  "- HMI Input - Exit 2 Select" %

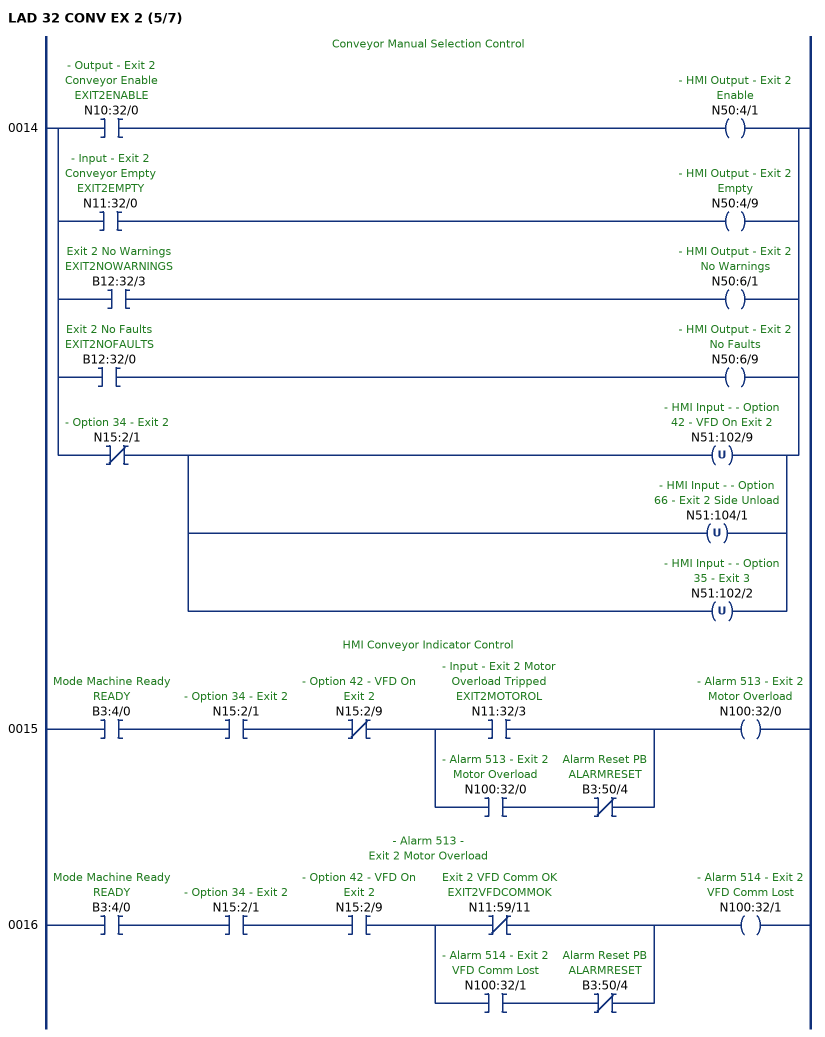
% Rung: 14 %
% Conveyor Manual Selection Control %
SOR BST XIC N10:32/0 OTE N50:4/1 NXB XIC N11:32/0 OTE N50:4/9 NXB XIC B12:32/3 OTE N50:6/1 NXB XIC B12:32/0 OTE N50:6/9 NXB XIO N15:2/1 BST OTU N51:102/9 NXB OTU N51:104/1 NXB OTU N51:102/2 BND BND EOR
%   N10:32/0  EXIT2ENABLE  "- Output - Exit 2 Conveyor Enable" %
%   N50:4/1  "- HMI Output - Exit 2 Enable" %
%   N11:32/0  EXIT2EMPTY  "- Input - Exit 2 Conveyor Empty" %
%   N50:4/9  "- HMI Output - Exit 2 Empty" %
%   B12:32/3  EXIT2NOWARNINGS  "Exit 2 No Warnings" %
%   N50:6/1  "- HMI Output - Exit 2 No Warnings" %
%   B12:32/0  EXIT2NOFAULTS  "Exit 2 No Faults" %
%   N50:6/9  "- HMI Output - Exit 2 No Faults" %
%   N15:2/1  "- Option 34 - Exit 2" %
%   N51:102/9  "- HMI Input - - Option 42 - VFD On Exit 2" %
%   N51:104/1  "- HMI Input - - Option 66 - Exit 2 Side Unload" %
%   N51:102/2  "- HMI Input - - Option 35 - Exit 3" %
% Rung: 15 %
% HMI Conveyor Indicator Control %
SOR XIC B3:4/0 XIC N15:2/1 XIO N15:2/9 BST XIC N11:32/3 NXB XIC N100:32/0 XIO B3:50/4 BND OTE N100:32/0 EOR
%   B3:4/0  READY  "Mode Machine Ready" %
%   N15:2/1  "- Option 34 - Exit 2" %
%   N15:2/9  "- Option 42 - VFD On Exit 2" %
%   N11:32/3  EXIT2MOTOROL  "- Input - Exit 2 Motor Overload Tripped" %
%   N100:32/0  "- Alarm 513 - Exit 2 Motor Overload" %
%   B3:50/4  ALARMRESET  "Alarm Reset PB" %
% Rung: 16 %
% - Alarm 513 -
% 
% Exit 2 Motor Overload %
SOR XIC B3:4/0 XIC N15:2/1 XIC N15:2/9 BST XIO N11:59/11 NXB XIC N100:32/1 XIO B3:50/4 BND OTE N100:32/1 EOR
%   B3:4/0  READY  "Mode Machine Ready" %
%   N15:2/1  "- Option 34 - Exit 2" %
%   N15:2/9  "- Option 42 - VFD On Exit 2" %
%   N11:59/11  EXIT2VFDCOMMOK  "Exit 2 VFD Comm OK" %
%   N100:32/1  "- Alarm 514 - Exit 2 VFD Comm Lost" %
%   B3:50/4  ALARMRESET  "Alarm Reset PB" %

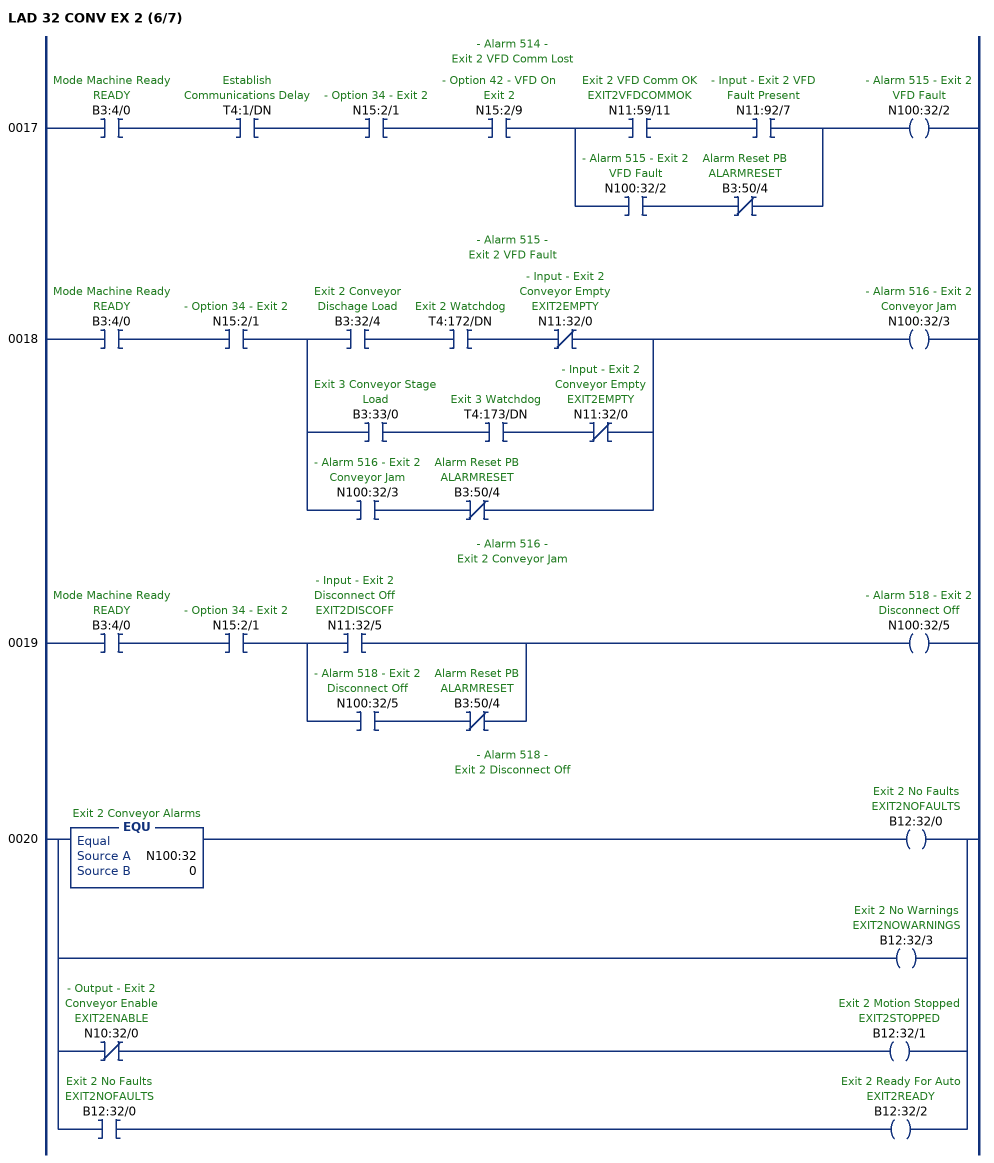
% Rung: 17 %
% - Alarm 514 -
% 
% Exit 2 VFD Comm Lost %
SOR XIC B3:4/0 XIC T4:1/DN XIC N15:2/1 XIC N15:2/9 BST XIC N11:59/11 XIC N11:92/7 NXB XIC N100:32/2 XIO B3:50/4 BND OTE N100:32/2 EOR
%   B3:4/0  READY  "Mode Machine Ready" %
%   T4:1  "Establish Communications Delay" %
%   N15:2/1  "- Option 34 - Exit 2" %
%   N15:2/9  "- Option 42 - VFD On Exit 2" %
%   N11:59/11  EXIT2VFDCOMMOK  "Exit 2 VFD Comm OK" %
%   N11:92/7  "- Input - Exit 2 VFD Fault Present" %
%   N100:32/2  "- Alarm 515 - Exit 2 VFD Fault" %
%   B3:50/4  ALARMRESET  "Alarm Reset PB" %
% Rung: 18 %
% - Alarm 515 -
% 
% Exit 2 VFD Fault %
SOR XIC B3:4/0 XIC N15:2/1 BST XIC B3:32/4 XIC T4:172/DN XIO N11:32/0 NXB XIC B3:33/0 XIC T4:173/DN XIO N11:32/0 NXB XIC N100:32/3 XIO B3:50/4 BND OTE N100:32/3 EOR
%   B3:4/0  READY  "Mode Machine Ready" %
%   N15:2/1  "- Option 34 - Exit 2" %
%   B3:32/4  "Exit 2 Conveyor Dischage Load" %
%   T4:172  "Exit 2 Watchdog" %
%   N11:32/0  EXIT2EMPTY  "- Input - Exit 2 Conveyor Empty" %
%   B3:33/0  "Exit 3 Conveyor Stage Load" %
%   T4:173  "Exit 3 Watchdog" %
%   N100:32/3  "- Alarm 516 - Exit 2 Conveyor Jam" %
%   B3:50/4  ALARMRESET  "Alarm Reset PB" %
% Rung: 19 %
% - Alarm 516 -
% 
% Exit 2 Conveyor Jam %
SOR XIC B3:4/0 XIC N15:2/1 BST XIC N11:32/5 NXB XIC N100:32/5 XIO B3:50/4 BND OTE N100:32/5 EOR
%   B3:4/0  READY  "Mode Machine Ready" %
%   N15:2/1  "- Option 34 - Exit 2" %
%   N11:32/5  EXIT2DISCOFF  "- Input - Exit 2 Disconnect Off" %
%   N100:32/5  "- Alarm 518 - Exit 2 Disconnect Off" %
%   B3:50/4  ALARMRESET  "Alarm Reset PB" %
% Rung: 20 %
% - Alarm 518 -
% 
% Exit 2 Disconnect Off %
SOR BST EQU N100:32 0 OTE B12:32/0 NXB OTE B12:32/3 NXB XIO N10:32/0 OTE B12:32/1 NXB XIC B12:32/0 OTE B12:32/2 BND EOR
%   N100:32  "Exit 2 Conveyor Alarms" %
%   B12:32/0  EXIT2NOFAULTS  "Exit 2 No Faults" %
%   B12:32/3  EXIT2NOWARNINGS  "Exit 2 No Warnings" %
%   N10:32/0  EXIT2ENABLE  "- Output - Exit 2 Conveyor Enable" %
%   B12:32/1  EXIT2STOPPED  "Exit 2 Motion Stopped" %
%   B12:32/2  EXIT2READY  "Exit 2 Ready For Auto" %

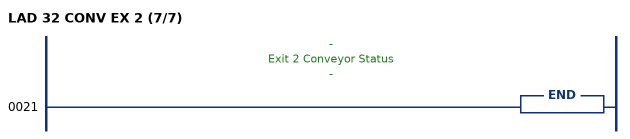
% Rung: 21 %
% -
% 
% Exit 2 Conveyor Status
% 
% - %
SOR END EOR

LADDER 33 "CONV EX 3"
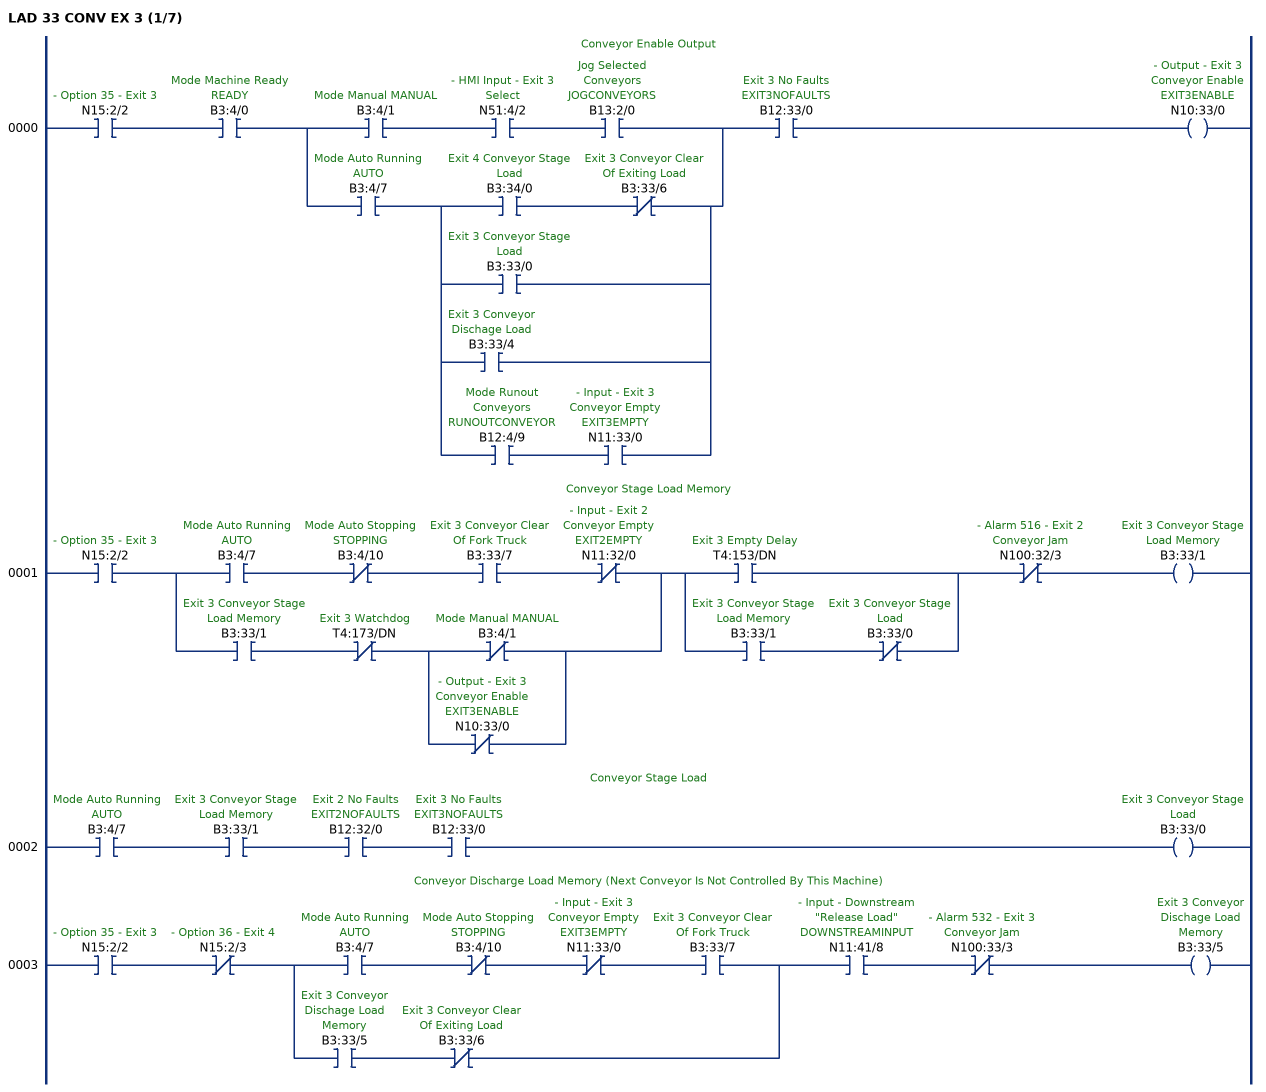
% Rung: 0 %
% Conveyor Enable Output %
SOR XIC N15:2/2 XIC B3:4/0 BST XIC B3:4/1 XIC N51:4/2 XIC B13:2/0 NXB XIC B3:4/7 BST XIC B3:34/0 XIO B3:33/6 NXB XIC B3:33/0 NXB XIC B3:33/4 NXB XIC B12:4/9 XIC N11:33/0 BND BND XIC B12:33/0 OTE N10:33/0 EOR
%   N15:2/2  "- Option 35 - Exit 3" %
%   B3:4/0  READY  "Mode Machine Ready" %
%   B3:4/1  MANUAL  "Mode Manual" %
%   N51:4/2  "- HMI Input - Exit 3 Select" %
%   B13:2/0  JOGCONVEYORS  "Jog Selected Conveyors" %
%   B3:4/7  AUTO  "Mode Auto Running" %
%   B3:34/0  "Exit 4 Conveyor Stage Load" %
%   B3:33/6  "Exit 3 Conveyor Clear Of Exiting Load" %
%   B3:33/0  "Exit 3 Conveyor Stage Load" %
%   B3:33/4  "Exit 3 Conveyor Dischage Load" %
%   B12:4/9  RUNOUTCONVEYOR  "Mode Runout Conveyors" %
%   N11:33/0  EXIT3EMPTY  "- Input - Exit 3 Conveyor Empty" %
%   B12:33/0  EXIT3NOFAULTS  "Exit 3 No Faults" %
%   N10:33/0  EXIT3ENABLE  "- Output - Exit 3 Conveyor Enable" %
% Rung: 1 %
% Conveyor Stage Load Memory %
SOR XIC N15:2/2 BST XIC B3:4/7 XIO B3:4/10 XIC B3:33/7 XIO N11:32/0 NXB XIC B3:33/1 XIO T4:173/DN BST XIO B3:4/1 NXB XIO N10:33/0 BND BND BST XIC T4:153/DN NXB XIC B3:33/1 XIO B3:33/0 BND XIO N100:32/3 OTE B3:33/1 EOR
%   N15:2/2  "- Option 35 - Exit 3" %
%   B3:4/7  AUTO  "Mode Auto Running" %
%   B3:4/10  STOPPING  "Mode Auto Stopping" %
%   B3:33/7  "Exit 3 Conveyor Clear Of Fork Truck" %
%   N11:32/0  EXIT2EMPTY  "- Input - Exit 2 Conveyor Empty" %
%   B3:33/1  "Exit 3 Conveyor Stage Load Memory" %
%   T4:173  "Exit 3 Watchdog" %
%   B3:4/1  MANUAL  "Mode Manual" %
%   N10:33/0  EXIT3ENABLE  "- Output - Exit 3 Conveyor Enable" %
%   T4:153  "Exit 3 Empty Delay" %
%   B3:33/0  "Exit 3 Conveyor Stage Load" %
%   N100:32/3  "- Alarm 516 - Exit 2 Conveyor Jam" %
% Rung: 2 %
% Conveyor Stage Load %
SOR XIC B3:4/7 XIC B3:33/1 XIC B12:32/0 XIC B12:33/0 OTE B3:33/0 EOR
%   B3:4/7  AUTO  "Mode Auto Running" %
%   B3:33/1  "Exit 3 Conveyor Stage Load Memory" %
%   B12:32/0  EXIT2NOFAULTS  "Exit 2 No Faults" %
%   B12:33/0  EXIT3NOFAULTS  "Exit 3 No Faults" %
%   B3:33/0  "Exit 3 Conveyor Stage Load" %
% Rung: 3 %
% Conveyor Discharge Load Memory (Next Conveyor Is Not Controlled By This Machine) %
SOR XIC N15:2/2 XIO N15:2/3 BST XIC B3:4/7 XIO B3:4/10 XIO N11:33/0 XIC B3:33/7 NXB XIC B3:33/5 XIO B3:33/6 BND XIC N11:41/8 XIO N100:33/3 OTE B3:33/5 EOR
%   N15:2/2  "- Option 35 - Exit 3" %
%   N15:2/3  "- Option 36 - Exit 4" %
%   B3:4/7  AUTO  "Mode Auto Running" %
%   B3:4/10  STOPPING  "Mode Auto Stopping" %
%   N11:33/0  EXIT3EMPTY  "- Input - Exit 3 Conveyor Empty" %
%   B3:33/7  "Exit 3 Conveyor Clear Of Fork Truck" %
%   B3:33/5  "Exit 3 Conveyor Dischage Load Memory" %
%   B3:33/6  "Exit 3 Conveyor Clear Of Exiting Load" %
%   N11:41/8  DOWNSTREAMINPUT  "- Input - Downstream "Release Load"" %
%   N100:33/3  "- Alarm 532 - Exit 3 Conveyor Jam" %

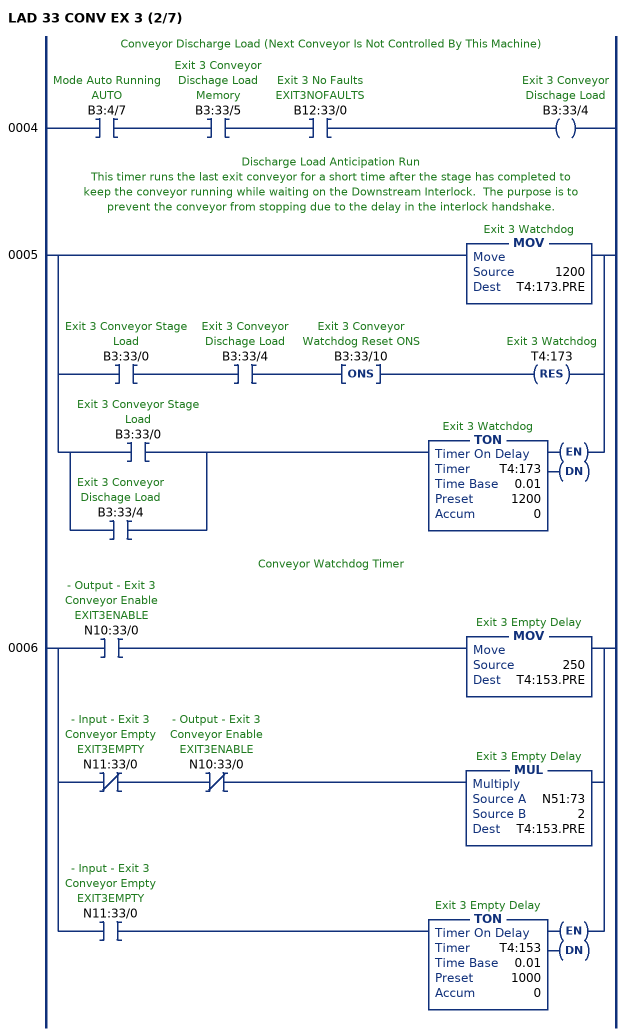
% Rung: 4 %
% Conveyor Discharge Load (Next Conveyor Is Not Controlled By This Machine) %
SOR XIC B3:4/7 XIC B3:33/5 XIC B12:33/0 OTE B3:33/4 EOR
%   B3:4/7  AUTO  "Mode Auto Running" %
%   B3:33/5  "Exit 3 Conveyor Dischage Load Memory" %
%   B12:33/0  EXIT3NOFAULTS  "Exit 3 No Faults" %
%   B3:33/4  "Exit 3 Conveyor Dischage Load" %
% Rung: 5 %
% Discharge Load Anticipation Run
% 
% This timer runs the last exit conveyor for a short time after the stage has completed to keep the conveyor running while waiting on the Downstream Interlock.  The purpose is to prevent the conveyor from stopping due to the delay in the interlock handshake. %
SOR BST MOV 1200 T4:173.PRE NXB XIC B3:33/0 XIC B3:33/4 ONS B3:33/10 RES T4:173 NXB BST XIC B3:33/0 NXB XIC B3:33/4 BND TON T4:173 0.01 1200 0 BND EOR
%   T4:173  "Exit 3 Watchdog" %
%   B3:33/0  "Exit 3 Conveyor Stage Load" %
%   B3:33/4  "Exit 3 Conveyor Dischage Load" %
%   B3:33/10  "Exit 3 Conveyor Watchdog Reset ONS" %
% Rung: 6 %
% Conveyor Watchdog Timer %
SOR BST XIC N10:33/0 MOV 250 T4:153.PRE NXB XIO N11:33/0 XIO N10:33/0 MUL N51:73 2 T4:153.PRE NXB XIC N11:33/0 TON T4:153 0.01 1000 0 BND EOR
%   N10:33/0  EXIT3ENABLE  "- Output - Exit 3 Conveyor Enable" %
%   T4:153  "Exit 3 Empty Delay" %
%   N11:33/0  EXIT3EMPTY  "- Input - Exit 3 Conveyor Empty" %
%   N51:73  "- HMI Input - Preset Truck Clear" %

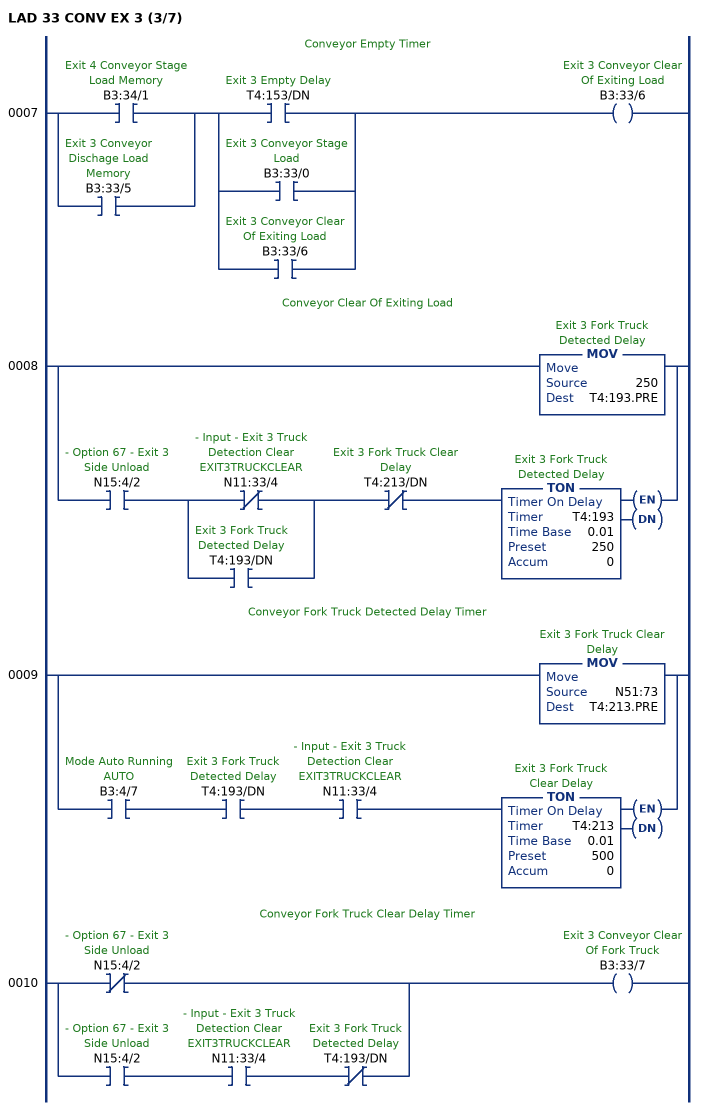
% Rung: 7 %
% Conveyor Empty Timer %
SOR BST XIC B3:34/1 NXB XIC B3:33/5 BND BST XIC T4:153/DN NXB XIC B3:33/0 NXB XIC B3:33/6 BND OTE B3:33/6 EOR
%   B3:34/1  "Exit 4 Conveyor Stage Load Memory" %
%   B3:33/5  "Exit 3 Conveyor Dischage Load Memory" %
%   T4:153  "Exit 3 Empty Delay" %
%   B3:33/0  "Exit 3 Conveyor Stage Load" %
%   B3:33/6  "Exit 3 Conveyor Clear Of Exiting Load" %
% Rung: 8 %
% Conveyor Clear Of Exiting Load %
SOR BST MOV 250 T4:193.PRE NXB XIC N15:4/2 BST XIO N11:33/4 NXB XIC T4:193/DN BND XIO T4:213/DN TON T4:193 0.01 250 0 BND EOR
%   T4:193  "Exit 3 Fork Truck Detected Delay" %
%   N15:4/2  "- Option 67 - Exit 3 Side Unload" %
%   N11:33/4  EXIT3TRUCKCLEAR  "- Input - Exit 3 Truck Detection Clear" %
%   T4:213  "Exit 3 Fork Truck Clear Delay" %
% Rung: 9 %
% Conveyor Fork Truck Detected Delay Timer %
SOR BST MOV N51:73 T4:213.PRE NXB XIC B3:4/7 XIC T4:193/DN XIC N11:33/4 TON T4:213 0.01 500 0 BND EOR
%   N51:73  "- HMI Input - Preset Truck Clear" %
%   T4:213  "Exit 3 Fork Truck Clear Delay" %
%   B3:4/7  AUTO  "Mode Auto Running" %
%   T4:193  "Exit 3 Fork Truck Detected Delay" %
%   N11:33/4  EXIT3TRUCKCLEAR  "- Input - Exit 3 Truck Detection Clear" %
% Rung: 10 %
% Conveyor Fork Truck Clear Delay Timer %
SOR BST XIO N15:4/2 NXB XIC N15:4/2 XIC N11:33/4 XIO T4:193/DN BND OTE B3:33/7 EOR
%   N15:4/2  "- Option 67 - Exit 3 Side Unload" %
%   N11:33/4  EXIT3TRUCKCLEAR  "- Input - Exit 3 Truck Detection Clear" %
%   T4:193  "Exit 3 Fork Truck Detected Delay" %
%   B3:33/7  "Exit 3 Conveyor Clear Of Fork Truck" %

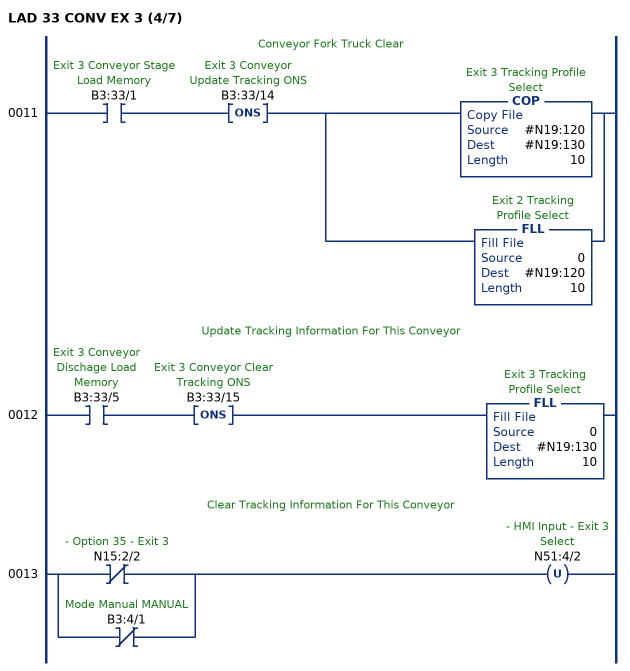
% Rung: 11 %
% Conveyor Fork Truck Clear %
SOR XIC B3:33/1 ONS B3:33/14 BST COP #N19:120 #N19:130 10 NXB FLL 0 #N19:120 10 BND EOR
%   B3:33/1  "Exit 3 Conveyor Stage Load Memory" %
%   B3:33/14  "Exit 3 Conveyor Update Tracking ONS" %
%   N19:120  "Exit 2 Tracking Profile Select" %
%   N19:130  "Exit 3 Tracking Profile Select" %
% Rung: 12 %
% Update Tracking Information For This Conveyor %
SOR XIC B3:33/5 ONS B3:33/15 FLL 0 #N19:130 10 EOR
%   B3:33/5  "Exit 3 Conveyor Dischage Load Memory" %
%   B3:33/15  "Exit 3 Conveyor Clear Tracking ONS" %
%   N19:130  "Exit 3 Tracking Profile Select" %
% Rung: 13 %
% Clear Tracking Information For This Conveyor %
SOR BST XIO N15:2/2 NXB XIO B3:4/1 BND OTU N51:4/2 EOR
%   N15:2/2  "- Option 35 - Exit 3" %
%   B3:4/1  MANUAL  "Mode Manual" %
%   N51:4/2  "- HMI Input - Exit 3 Select" %

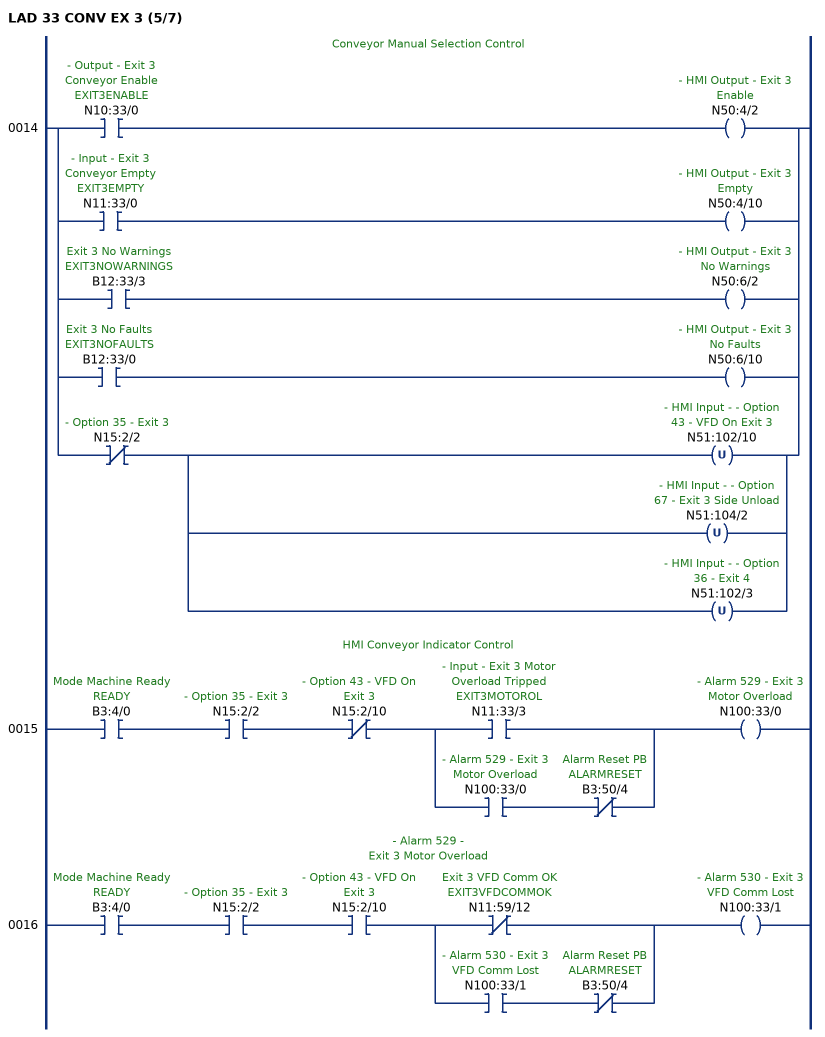
% Rung: 14 %
% Conveyor Manual Selection Control %
SOR BST XIC N10:33/0 OTE N50:4/2 NXB XIC N11:33/0 OTE N50:4/10 NXB XIC B12:33/3 OTE N50:6/2 NXB XIC B12:33/0 OTE N50:6/10 NXB XIO N15:2/2 BST OTU N51:102/10 NXB OTU N51:104/2 NXB OTU N51:102/3 BND BND EOR
%   N10:33/0  EXIT3ENABLE  "- Output - Exit 3 Conveyor Enable" %
%   N50:4/2  "- HMI Output - Exit 3 Enable" %
%   N11:33/0  EXIT3EMPTY  "- Input - Exit 3 Conveyor Empty" %
%   N50:4/10  "- HMI Output - Exit 3 Empty" %
%   B12:33/3  EXIT3NOWARNINGS  "Exit 3 No Warnings" %
%   N50:6/2  "- HMI Output - Exit 3 No Warnings" %
%   B12:33/0  EXIT3NOFAULTS  "Exit 3 No Faults" %
%   N50:6/10  "- HMI Output - Exit 3 No Faults" %
%   N15:2/2  "- Option 35 - Exit 3" %
%   N51:102/10  "- HMI Input - - Option 43 - VFD On Exit 3" %
%   N51:104/2  "- HMI Input - - Option 67 - Exit 3 Side Unload" %
%   N51:102/3  "- HMI Input - - Option 36 - Exit 4" %
% Rung: 15 %
% HMI Conveyor Indicator Control %
SOR XIC B3:4/0 XIC N15:2/2 XIO N15:2/10 BST XIC N11:33/3 NXB XIC N100:33/0 XIO B3:50/4 BND OTE N100:33/0 EOR
%   B3:4/0  READY  "Mode Machine Ready" %
%   N15:2/2  "- Option 35 - Exit 3" %
%   N15:2/10  "- Option 43 - VFD On Exit 3" %
%   N11:33/3  EXIT3MOTOROL  "- Input - Exit 3 Motor Overload Tripped" %
%   N100:33/0  "- Alarm 529 - Exit 3 Motor Overload" %
%   B3:50/4  ALARMRESET  "Alarm Reset PB" %
% Rung: 16 %
% - Alarm 529 -
% 
% Exit 3 Motor Overload %
SOR XIC B3:4/0 XIC N15:2/2 XIC N15:2/10 BST XIO N11:59/12 NXB XIC N100:33/1 XIO B3:50/4 BND OTE N100:33/1 EOR
%   B3:4/0  READY  "Mode Machine Ready" %
%   N15:2/2  "- Option 35 - Exit 3" %
%   N15:2/10  "- Option 43 - VFD On Exit 3" %
%   N11:59/12  EXIT3VFDCOMMOK  "Exit 3 VFD Comm OK" %
%   N100:33/1  "- Alarm 530 - Exit 3 VFD Comm Lost" %
%   B3:50/4  ALARMRESET  "Alarm Reset PB" %

